ACTION _800_Reset:
Axis[ID].aStop();
CASE RestStep OF
0:(***************复位命令**************************)
	IF GVL_API.stAxis[ID].reset OR GVL.Reset THEN
		GVL_API.stAxis[ID].initialize:=FALSE;
		GVL_API.stAxis[ID].homeExe:=FALSE; 
		GVL_API.stAxis[ID].stop:=FALSE;
		GVL_API.stAxis[ID].JogBackwards:=FALSE;
		GVL_API.stAxis[ID].JogForward:=FALSE;
		GVL_API.stAxis[ID].MoveAbsoluteExe:=FALSE;
		GVL_API.stAxis[ID].MoveConstantVelocity:=FALSE;
		GVL_API.stAxis[ID].MoveRelativeExe:=FALSE;
		GVL_API.stAxis[ID].velocity:=0;
		GVL_API.stAxis[ID].requestedoffset:=0;
		GVL_API.stAxis[ID].requestedposition:=0;
		GVL_API.stAxis[ID].constantvelocitystart:=0;
		GVL_API.stAxis[ID].constanvelocityend:=0;
		FB_Home(ref:=Axis[ID].Ref , Execute:= FALSE);
		GVL_API.stAxis[ID].Home_Done:=FALSE;
		GVL_API.stAxis[ID].Move_Done:=FALSE;
		RestStep:=1;
	END_IF
1:	
		RestStep:=2;

2:(***************EORROR来的错误**************************)
		GVL_API.stAxis[ID].reset:=FALSE;
		parameter_out_of_range:=FALSE;
		SpeedNotReach:=FALSE;		
		RestStep:=20;
	
10:	(***************轴错误复位**************************)		
		Axis[ID].Reset_do:=TRUE;		
		RestStep:=100;		
20:	(***************轴停止*****************************)
		Axis[ID].aStop(stop_do:=TRUE);		
		RestStep:=30;
30:
	IF  Axis[ID].Ref.Status.NotMoving   THEN 		
		RestStep:=10;	
	END_IF
100:		
	IF Axis[ID].Ref.Status.NotMoving THEN 
		Axis[Id].aPower(power_do:=FALSE);
		GVL_API.stAxis[ID].Error:=FALSE;
		GVL_API.stAxis[ID].state:=AxisStateEnum.off;
		GVL_API.stAxis[ID].Errorid:=Axis_XY_ErrorEnum.no_error;
			SysStep:=0;
			RestStep:=0;
	END_IF
	  
END_CASE
END_ACTION

ACTION ACT_LOG:
(*************************LOG*******************************************)
log_ID:=100;
//initialize
AlarmActionArray[log_ID+1].AlarmMsg.EN	:=	'Fast Scan Initialize cmdtimeout:';
AlarmActionArray[log_ID+1].AlarmMsg.EN	:=CONCAT(AlarmActionArray[log_ID+1].AlarmMsg.EN,
																	LREAL_TO_STRING(GVL_API.stAxis[ID].commandtimeout));
AlarmActionArray[log_ID+1].AlarmMsg.EN	:=CONCAT(AlarmActionArray[log_ID+1].AlarmMsg.EN,'; velocity:');
AlarmActionArray[log_ID+1].AlarmMsg.EN	:=CONCAT(AlarmActionArray[log_ID+1].AlarmMsg.EN,
																	LREAL_TO_STRING(GVL_API.stAxis[ID].velocity));	
AlarmActionArray[log_ID+1].AlarmMsg.EN	:=CONCAT(AlarmActionArray[log_ID+1].AlarmMsg.EN,'; acce:');																
AlarmActionArray[log_ID+1].AlarmMsg.EN	:=CONCAT(AlarmActionArray[log_ID+1].AlarmMsg.EN,
																	LREAL_TO_STRING(GVL_API.stAxis[ID].acceleration));
AlarmActionArray[log_ID+1].AlarmMsg.EN	:=CONCAT(AlarmActionArray[log_ID+1].AlarmMsg.EN,'; maxposition:');	
AlarmActionArray[log_ID+1].AlarmMsg.EN	:=CONCAT(AlarmActionArray[log_ID+1].AlarmMsg.EN,
																	LREAL_TO_STRING(GVL_API.stAxis[ID].maxDistance));
fbSetAlarm[log_ID+1](
	InUse:=TRUE , 
	//EventId:=log_ID+1 , 
	EventActive:=GVL_API.stAxis[ID].initialize , 
	EventClass:=Alm_EventClass.Event , 
	ToTheLogFile:=TRUE, 
	ToTheHistory:=TRUE , 
 );
 //home
AlarmActionArray[log_ID+2].AlarmMsg.EN	:=	'Fast Scan Home homingvelocity:';
AlarmActionArray[log_ID+2].AlarmMsg.EN	:=CONCAT(AlarmActionArray[log_ID+2].AlarmMsg.EN,
																	LREAL_TO_STRING(GVL_API.stAxis[ID].homingvelocity));
AlarmActionArray[log_ID+2].AlarmMsg.EN	:=CONCAT(AlarmActionArray[log_ID+2].AlarmMsg.EN,'; homeoffset:');
AlarmActionArray[log_ID+2].AlarmMsg.EN	:=CONCAT(AlarmActionArray[log_ID+2].AlarmMsg.EN,
																	LREAL_TO_STRING(GVL_API.stAxis[ID].homeoffset));		
AlarmActionArray[log_ID+2].AlarmMsg.EN	:=CONCAT(AlarmActionArray[log_ID+2].AlarmMsg.EN,'; homingtimeout:');
AlarmActionArray[log_ID+2].AlarmMsg.EN	:=CONCAT(AlarmActionArray[log_ID+2].AlarmMsg.EN,
																	LREAL_TO_STRING(GVL_API.stAxis[ID].homingtimeout));																
fbSetAlarm[log_ID+2](
	InUse:=TRUE , 
	//EventId:=log_ID+2 , 
	EventActive:=GVL_API.stAxis[ID].homeExe , 
	EventClass:=Alm_EventClass.Event , 
	ToTheLogFile:=TRUE, 
	ToTheHistory:=TRUE , 
 );
 //MoveRelative
AlarmActionArray[log_ID+3].AlarmMsg.EN	:=CONCAT('Fast Scan MoveRelative displacement:',
																	LREAL_TO_STRING(GVL_API.stAxis[ID].requestedoffset));
AlarmActionArray[log_ID+3].AlarmMsg.EN	:=CONCAT(AlarmActionArray[log_ID+3].AlarmMsg.EN,'; velocity:');
AlarmActionArray[log_ID+3].AlarmMsg.EN	:=CONCAT(AlarmActionArray[log_ID+3].AlarmMsg.EN,
																	LREAL_TO_STRING(GVL_API.stAxis[ID].velocity));
AlarmActionArray[log_ID+3].AlarmMsg.EN	:=CONCAT(AlarmActionArray[log_ID+3].AlarmMsg.EN,'; acc:');
AlarmActionArray[log_ID+3].AlarmMsg.EN	:=CONCAT(AlarmActionArray[log_ID+3].AlarmMsg.EN,
																	LREAL_TO_STRING(GVL_API.stAxis[ID].acceleration));
AlarmActionArray[log_ID+3].AlarmMsg.EN	:=CONCAT(AlarmActionArray[log_ID+3].AlarmMsg.EN,'; jerk:');																	
AlarmActionArray[log_ID+3].AlarmMsg.EN	:=CONCAT(AlarmActionArray[log_ID+3].AlarmMsg.EN,
																	LREAL_TO_STRING(GVL_API.stAxis[ID].jerk));
fbSetAlarm[log_ID+3](
	InUse:=TRUE , 
	//EventId:=log_ID+3 , 
	EventActive:=GVL_API.stAxis[ID].MoveRelativeExe , 
	EventClass:=Alm_EventClass.Event , 
	ToTheLogFile:=TRUE, 
	ToTheHistory:=TRUE , 
 );
 //MoveAbsoluteExe
AlarmActionArray[log_ID+4].AlarmMsg.EN	:=CONCAT('Fast Scan MoveAbsolute position:',
																	LREAL_TO_STRING(GVL_API.stAxis[ID].requestedposition));
AlarmActionArray[log_ID+4].AlarmMsg.EN	:=CONCAT(AlarmActionArray[log_ID+4].AlarmMsg.EN,'; velocity:');
AlarmActionArray[log_ID+4].AlarmMsg.EN	:=CONCAT(AlarmActionArray[log_ID+4].AlarmMsg.EN,
																	LREAL_TO_STRING(GVL_API.stAxis[ID].velocity));
AlarmActionArray[log_ID+4].AlarmMsg.EN	:=CONCAT(AlarmActionArray[log_ID+4].AlarmMsg.EN,'; acc:');
AlarmActionArray[log_ID+4].AlarmMsg.EN	:=CONCAT(AlarmActionArray[log_ID+4].AlarmMsg.EN,
																	LREAL_TO_STRING(GVL_API.stAxis[ID].acceleration));
AlarmActionArray[log_ID+4].AlarmMsg.EN	:=CONCAT(AlarmActionArray[log_ID+4].AlarmMsg.EN,'; jerk:');																	
AlarmActionArray[log_ID+4].AlarmMsg.EN	:=CONCAT(AlarmActionArray[log_ID+4].AlarmMsg.EN,
																	LREAL_TO_STRING(GVL_API.stAxis[ID].jerk));
fbSetAlarm[log_ID+4](
	InUse:=TRUE , 
	//EventId:=log_ID+4 , 
	EventActive:=GVL_API.stAxis[ID].MoveAbsoluteExe , 
	EventClass:=Alm_EventClass.Event , 
	ToTheLogFile:=TRUE, 
	ToTheHistory:=TRUE , 
 );
 //MoveConstantVelocity
AlarmActionArray[log_ID+5].AlarmMsg.EN	:=CONCAT('Fast Scan MoveConstantVelocity,',
																LREAL_TO_STRING(GVL_API.stAxis[ID].constantvelocitystart));
AlarmActionArray[log_ID+5].AlarmMsg.EN	:=CONCAT(AlarmActionArray[log_ID+5].AlarmMsg.EN,'->');
AlarmActionArray[log_ID+5].AlarmMsg.EN	:=CONCAT(AlarmActionArray[log_ID+5].AlarmMsg.EN,
																LREAL_TO_STRING(GVL_API.stAxis[ID].constanvelocityend));
AlarmActionArray[log_ID+5].AlarmMsg.EN	:=CONCAT(AlarmActionArray[log_ID+5].AlarmMsg.EN,'->');
AlarmActionArray[log_ID+5].AlarmMsg.EN	:=CONCAT(AlarmActionArray[log_ID+5].AlarmMsg.EN,
																LREAL_TO_STRING(GVL_API.stAxis[ID].requestedposition));
AlarmActionArray[log_ID+5].AlarmMsg.EN	:=CONCAT(AlarmActionArray[log_ID+5].AlarmMsg.EN,'; velocity:');
AlarmActionArray[log_ID+5].AlarmMsg.EN	:=CONCAT(AlarmActionArray[log_ID+5].AlarmMsg.EN,
																	LREAL_TO_STRING(GVL_API.stAxis[ID].velocity));
AlarmActionArray[log_ID+5].AlarmMsg.EN	:=CONCAT(AlarmActionArray[log_ID+5].AlarmMsg.EN,'; acc:');
AlarmActionArray[log_ID+5].AlarmMsg.EN	:=CONCAT(AlarmActionArray[log_ID+5].AlarmMsg.EN,
																	LREAL_TO_STRING(GVL_API.stAxis[ID].acceleration));
AlarmActionArray[log_ID+5].AlarmMsg.EN	:=CONCAT(AlarmActionArray[log_ID+5].AlarmMsg.EN,'; jerk:');																	
AlarmActionArray[log_ID+5].AlarmMsg.EN	:=CONCAT(AlarmActionArray[log_ID+5].AlarmMsg.EN,
																	LREAL_TO_STRING(GVL_API.stAxis[ID].jerk));
fbSetAlarm[log_ID+5](
	InUse:=TRUE , 
	//EventId:=log_ID+5 , 
	EventActive:=GVL_API.stAxis[ID].MoveConstantVelocity , 
	EventClass:=Alm_EventClass.Event , 
	ToTheLogFile:=TRUE, 
	ToTheHistory:=TRUE , 
 );
//stop
AlarmActionArray[log_ID+6].AlarmMsg.EN	:=	'Fast Scan MoveStop ';
fbSetAlarm[log_ID+6](
	InUse:=TRUE , 
	//EventId:=log_ID+6 , 
	EventActive:=GVL_API.stAxis[ID].stop , 
	EventClass:=Alm_EventClass.Event , 
	ToTheLogFile:=TRUE, 
	ToTheHistory:=TRUE , 
 );
 //enabled
AlarmActionArray[log_ID+7].AlarmMsg.EN	:=	'Fast Scan Enabled ';
fbSetAlarm[log_ID+7](
	InUse:=TRUE , 
	//EventId:=log_ID+7 , 
	EventActive:=GVL_API.stAxis[ID].enabled , 
	EventClass:=Alm_EventClass.Event , 
	ToTheLogFile:=TRUE, 
	ToTheHistory:=TRUE , 
 );
  //disable
AlarmActionArray[log_ID+8].AlarmMsg.EN	:=	'Fast Scan Disable ';
fbSetAlarm[log_ID+8](
	InUse:=TRUE , 
	//EventId:=log_ID+8 , 
	EventActive:=GVL_API.stAxis[ID].Disable , 
	EventClass:=Alm_EventClass.Event , 
	ToTheLogFile:=TRUE, 
	ToTheHistory:=TRUE , 
 );
//ERROR,log_ErrorEnum只能等于一个常数
CASE GVL_API.stAxis[ID].errorid  OF
0	:	log_ErrorEnum	:=	0	;
1	:	log_ErrorEnum	:=	1	;
2	:	log_ErrorEnum	:=	2	;
3	:	log_ErrorEnum	:=	3	;
4	:	log_ErrorEnum	:=	4	;
5	:	log_ErrorEnum	:=	5	;
6	:	log_ErrorEnum	:=	6	;
7	:	log_ErrorEnum	:=	7	;
8	:	log_ErrorEnum	:=	8	;
9	:	log_ErrorEnum	:=	9	;
10	:	log_ErrorEnum	:=	10	;
11	:	log_ErrorEnum	:=	11	;
12	:	log_ErrorEnum	:=	12	;
13	:	log_ErrorEnum	:=	13	;
14	:	log_ErrorEnum	:=	14	;
15	:	log_ErrorEnum	:=	15	;
16	:	log_ErrorEnum	:=	16	;
666	:	log_ErrorEnum	:=	666	;

END_CASE

AlarmActionArray[log_ID+9].AlarmMsg.EN	:=CONCAT('Fast Scan Error: ',TO_STRING(log_ErrorEnum));
fbSetAlarm[log_ID+9](
	InUse:=TRUE , 
//	EventId:=log_ID+9 , 
	EventActive:=GVL_API.stAxis[ID].errorid<>0 AND GVL_API.stAxis[ID].errorid<>666 , 
	EventClass:=Alm_EventClass.Alarm , 
	ToTheLogFile:=TRUE, 
	ToTheHistory:=TRUE , 
 );
 
//reset
AlarmActionArray[log_ID+10].AlarmMsg.EN	:=	'Fast Scan Reset ';
fbSetAlarm[log_ID+10](
	InUse:=TRUE , 
	EventId:=log_ID+10 , 
	EventActive:=GVL_API.stAxis[ID].reset , 
	EventClass:=Alm_EventClass.Event , 
	ToTheLogFile:=TRUE, 
	ToTheHistory:=TRUE , 
 );
 //AXIX_ERRORID
 AlarmActionArray[log_ID+11].AlarmMsg.EN	:=CONCAT('Fast Scan Axis_ErrorID: ',
																		UDINT_TO_STRING(Axis[ID].Ref.Status.ErrorID));
fbSetAlarm[log_ID+11](
	InUse:=TRUE , 
	EventId:=log_ID+11 , 
	EventActive:=Axis[ID].Ref.Status.Error , 
	EventClass:=Alm_EventClass.Event , 
	ToTheLogFile:=TRUE, 
	ToTheHistory:=TRUE , 
 );
END_ACTION

ACTION ACT_Safety:
(*****************SAFETY******************************)
IF GVL_API.stAxis[ID].state<>AxisStateEnum.off AND  GVL_API.stAxis[ID].state<>AxisStateEnum.error THEN 
	IF GVl.Emstop_Button OR GVL.Emstop_SAFE  THEN 
		GVL_API.stAxis[ID].errorid:=Axis_XY_ErrorEnum.emergency_error;
		Axis[ID].aStop(stop_do:=TRUE,Dec:=HMI_EM_STOP_Dec_FS,Jerk:=HMI_EM_STOP_Jerk_FS);
		//Axis[ID].aStop(stop_do:=TRUE,Jerk:=GVL_API.stAxis[ID].jerk);
		SysStep:=700;
	ELSIF GVL.shuttle_crash OR  Axis[ID].IO.snLimitN OR Axis[ID].IO.snLimitP  THEN 	
		GVL_API.stAxis[ID].errorid:=Axis_XY_ErrorEnum.trigger_Limit;
		Axis[ID].aStop(stop_do:=TRUE,Dec:=HMI_EM_STOP_Dec_FS,Jerk:=HMI_EM_STOP_Jerk_FS);
		SysStep:=700;
	(*ELSIF GVL.interlock_triggered THEN 
		GVL_API.stAxis[ID].ErrorId:=Axis_XY_ErrorEnum.interlock_error;
		Axis[ID].aStop(stop_do:=TRUE,Dec:=HMI_EM_STOP_Dec_FS,Jerk:=HMI_EM_STOP_Jerk_FS);
		SysStep:=700;
	*)
	ELSIF  Axis[ID].mcReadStatus.ErrorID=18000 THEN 
		GVL_API.stAxis[ID].errorid:=Axis_XY_ErrorEnum.Drive_not_ready_for_operation;
		SysStep:=700;
	ELSIF   Axis[ID].mcReadStatus.ErrorID=17510 THEN 
		GVL_API.stAxis[ID].errorid:=Axis_XY_ErrorEnum.Invalid_IO_data_for_more_than_n_subsequent_NC_cycles_encoder;
		SysStep:=700;	
	ELSIF  Axis[ID].mcReadStatus.ErrorID<>0 THEN 
		GVL_API.stAxis[ID].errorid:=Axis[ID].mcReadStatus.ErrorID;
		SysStep:=700;
	//ELSE 
	//	GVL_API.stAxis[ID].error:=Axis_XY_ErrorEnum.no_error;
	//	SysStep:=700;			
	END_IF	
END_IF

(*****************AXIS_ERROR******************************)
GVL_API.stAxis[ID].AxisErrorId:=Axis[ID].Ref.Status.ErrorID;
END_ACTION

END_PROGRAM

// ---- POUs/010_Motion/MotionBase/FB_MoveFS_Exte.TcPOU
FUNCTION_BLOCK FB_MoveFS_Exte
VAR_INPUT
	enable	:BOOL;
	ref		:AXIS_REF;
	jogF	:BOOL;
	jogB	:BOOL;
	Move_Stop:BOOL;
	PosLimit			:BOOL;			(*正极限位信号*)
	NegLimit			:BOOL;			(*负极限位信号*)
	maxDistance			:LREAL;			(*最大行程*)
	Acceleration		:LREAL;
	Deceleration		:LREAL;
	Jerk				:LREAL;
END_VAR
VAR_OUTPUT	
END_VAR
VAR
	MC_Read:MC_ReadStatus;
	MC_ABS:MC_MoveAbsolute;
	MC_REL:MC_MoveRelative;
	MC_Jog:MC_Jog;
	
	MC_ABS1:MC_MoveAbsolute;

	step1,step2,step3		:INT;	
	R_TRIG1,R_TRIG2,R_TRIG3	:R_TRIG;
	R_TRIG_done				:R_TRIG;
	ton_NotMoving			:TON;
	ton_Moving				:TON;
	rel_do					:BOOL;
	abs_do					:BOOL;
	jogF_do					:BOOL;
	jogB_do					:BOOL;
	
	abs_do1    			    :BOOL;
	error					:BOOL;

	MoveAbsolute_Busy		:BOOL;
	MoveConstantVelocity_Busy:BOOL;
	MoveRelative_Busy		:BOOL;
	jog_EN					:BOOL;
	FB_START_r_trig:		R_TRIG;
	start					:BOOL;
	jog_f_trig				:F_TRIG;
	ton_NotMoving_r_trig:Tc2_Standard.R_TRIG;
	Positive_Direction:BOOL;//正向
	Negative_Direction:BOOL;//负向
	
END_VAR
VAR_IN_OUT 
	MoveRelExe					:BOOL;
	MoveAbsExe					:BOOL;
	MoveConstantVelocityExe		:BOOL;//
	Velo						:LREAL;	//mm/s
	TargetRel					:LREAL;//mm
	TargetAbs					:LREAL;//mm
	ConstantVelocityStart		:LREAL;//mm		The position to start moving with a constant velocity
												//      0 < ConstantVelocityStart< ConstanVelocityEnd< RequestedPosition
	ConstanVelocityEnd			:LREAL;//mm		The position to end moving with a constant velocity											
	Done						:BOOL;
	NotMovingTimeOut 			:BOOL;
	SpeedNotReach				:BOOL;
END_VAR

(*********************NOT MOVING TIMEOUT***************************)
FB_START_r_trig(CLK:=jogF OR jogB OR MoveRelExe OR MoveAbsExe OR MoveConstantVelocityExe  , Q=> );
IF FB_START_r_trig.Q THEN 
	start:=TRUE;
END_IF
ton_NotMoving(IN:=Ref.Status.NotMoving AND start  , PT:= T#5S, Q=> , ET=> );
ton_NotMoving_r_trig(CLK:=ton_NotMoving.Q , Q=> );
IF ton_NotMoving_r_trig.Q THEN 
		NotMovingTimeOut:=TRUE;	
END_IF

Call_FB();
JOG();
MoveAbsolute();
MoveConstantVelocity();
MoveRelative();


(*********************error***************************)
IF ton_NotMoving.Q OR error OR SpeedNotReach THEN	
	start:=FALSE;
	error:=FALSE;
	ton_NotMoving(IN:=FALSE);	
	step1:=step2:=step2:=0;	
	MoveRelExe:=FALSE;
	MoveAbsExe:=FALSE;
	MoveConstantVelocityExe:=FALSE;
	Velo:=0;
	TargetAbs:=0;
	TargetRel:=0;
	ConstantVelocityStart:=0;
	ConstanVelocityEnd:=0;
	step1:=step2:=step3:=0;
	R_TRIG1(CLK:=FALSE);
	R_TRIG2(CLK:=FALSE);
	R_TRIG3(CLK:=FALSE);
END_IF

(*********************move done***************************)
IF MoveAbsolute_Busy OR MoveConstantVelocity_Busy OR  MoveRelative_Busy THEN 
	Done:=FALSE;
	jogF:=FALSE;
	jogB:=FALSE;
END_IF

jog_f_trig(CLK:=jogB OR jogF , Q=> );

R_TRIG_done(CLK:=MC_REL.Done OR MC_ABS.Done OR MC_ABS1.Done  OR jog_f_trig.Q OR Move_Stop , Q=> );
IF R_TRIG_done.Q THEN 	
	start:=FALSE;
	R_TRIG_done(CLK:=FALSE);
	NotMovingTimeOut:=FALSE;
	ton_NotMoving(IN:=FALSE);
	step1:=step2:=step3:=0;	
	MoveRelExe:=FALSE;
	MoveAbsExe:=FALSE;
	MoveConstantVelocityExe:=FALSE;
	Velo:=0;
	TargetAbs:=0;
	TargetRel:=0;
	ConstantVelocityStart:=0;
	ConstanVelocityEnd:=0;
	Done:=TRUE ;
END_IF

ACTION Call_FB:
MC_Read(
	Axis:=ref , 
	Enable:=TRUE);
MC_REL(
	Axis:=ref , 
	Execute:=rel_do , 
	Distance:=TargetRel , 
	Velocity:=Velo , 
	Acceleration:=Acceleration , 
	Deceleration:=Deceleration , 
	Jerk:=Jerk , 
	BufferMode:= , 
	Options:= , 
	Done=> , 
	Busy=>MoveRelative_Busy , 
	Active=> , 
	CommandAborted=> , 
	Error=> , 
	ErrorID=> );
	IF MC_REL.Busy THEN 
		rel_do:=FALSE;
		MoveRelExe:=FALSE;
	END_IF
MC_ABS(
	Axis:=ref , 
	Execute:=abs_do , 
	Position:=TargetAbs , 
	Velocity:=Velo , 
	Acceleration:=Acceleration , 
	Deceleration:=Deceleration , 
	Jerk:=Jerk , 
	BufferMode:= , 
	Options:= , 
	Done=> , 
	Busy=>MoveAbsolute_Busy , 
	Active=> , 
	CommandAborted=> , 
	Error=> , 
	ErrorID=> );
	IF MC_ABS.Busy THEN 
		abs_do:=FALSE;
		MoveAbsExe:=FALSE;
	END_IF
MC_Jog(
	Axis:=ref , 
	JogForward:=jogF_do , 
	JogBackwards:=jogB_do , 
	Mode:=MC_JOGMODE_CONTINOUS , 
	Position:= , 
	Velocity:=Velo , 
	Acceleration:=Acceleration , 
	Deceleration:=Deceleration , 
	Jerk:=Jerk , 
	Done=> , 
	Busy=> , 
	Active=> , 
	CommandAborted=> , 
	Error=> , 
	ErrorID=> );
MC_ABS1(
	Axis:=ref , 
	Execute:=abs_do1 , 
	Position:=TargetAbs , 
	Velocity:=Velo , 
	Acceleration:=Acceleration , 
	Deceleration:=Deceleration , 
	Jerk:=Jerk , 
	BufferMode:= , 
	Options:= , 
	Done=> , 
	Busy=> , 
	Active=> , 
	CommandAborted=> , 
	Error=> , 
	ErrorID=> );
	IF MC_ABS1.Busy THEN 
		abs_do1:=FALSE;
		MoveConstantVelocityExe:=FALSE;
	END_IF
END_ACTION

ACTION JOG:
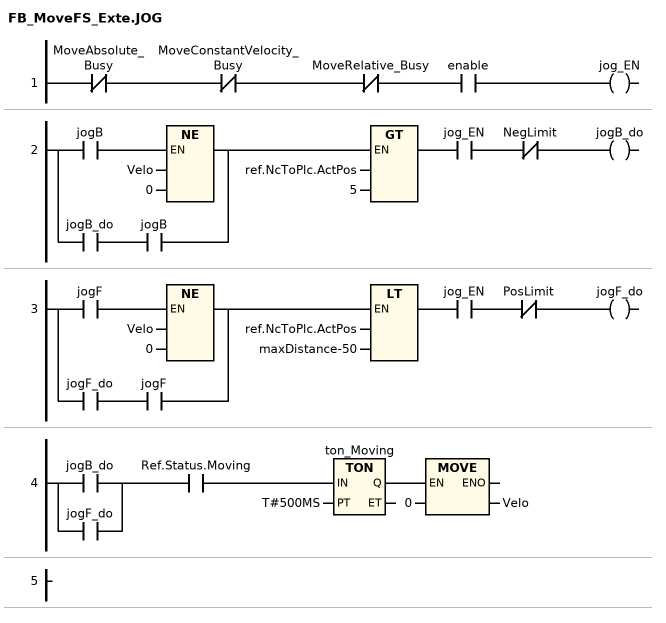
// NETWORK 1
jog_EN := NOT MoveAbsolute_Busy AND NOT MoveConstantVelocity_Busy AND NOT MoveRelative_Busy AND enable;

// NETWORK 2
jogB_do := ((jogB AND Velo <> 0 OR jogB_do AND jogB) AND ref.NcToPlc.ActPos > 5) AND jog_EN AND NOT NegLimit;

// NETWORK 3
jogF_do := ((jogF AND Velo <> 0 OR jogF_do AND jogF) AND ref.NcToPlc.ActPos < (maxDistance-50)) AND jog_EN AND NOT PosLimit;

// NETWORK 4
ton_Moving(IN := (jogB_do OR jogF_do) AND Ref.Status.Moving, PT := T#500MS); // TON
IF ton_Moving.Q THEN Velo := 0; END_IF

// NETWORK 5
END_ACTION

ACTION MoveAbsolute:
(****************ABS********************)
R_TRIG2(CLK:=MoveAbsExe AND Ref.Status.NotMoving AND enable   , Q=> );

CASE step2 OF 
	0:				
		IF R_TRIG2.Q THEN 
			R_TRIG2(CLK:=FALSE);			
			MoveAbsExe:=FALSE;
			step2:=1;
		END_IF
	1:	
		IF   Velo<>0 THEN 		
			abs_do:=TRUE;
			step2:=2;
		END_IF
	2:
		IF MC_ABS.Busy THEN 
			abs_do:=FALSE;								
			step2 :=0;
		END_IF	
END_CASE


IF  MoveAbsolute_Busy THEN 
	MoveRelExe:=FALSE;
	MoveConstantVelocityExe:=FALSE;
END_IF
END_ACTION

ACTION MoveConstantVelocity:
(****************MoveConstantVelocity********************)
R_TRIG3(CLK:=MoveConstantVelocityExe AND Ref.Status.NotMoving AND enable  , Q=> );
CASE step3 OF 
	0:				
		IF R_TRIG3.Q THEN 
			R_TRIG3(CLK:=FALSE);
			abs_do1:=FALSE;		
			MoveConstantVelocityExe:=FALSE;
			step3:=1;
		END_IF
	1:	//
		IF   Velo<>0 THEN 		
			abs_do1:=TRUE;
			step3:=2;
		END_IF
		
	2:	//启动第二段，匀速段,增加到达位置时速度判断
		IF ConstanVelocityEnd>ConstantVelocityStart THEN 
			Positive_Direction:=TRUE;
			Negative_Direction:=FALSE;
		ELSE
			Positive_Direction:=FALSE;
			Negative_Direction:=TRUE;	
		END_IF

			
		IF 	(Positive_Direction AND ref.NcToPlc.ActPos>=ConstantVelocityStart ) OR 
			(Negative_Direction AND ref.NcToPlc.ActPos<=ConstantVelocityStart ) THEN 
			
			 IF ABS(ABS(ref.NcToPlc.ActVelo)-Velo)<=30 THEN
				step3 :=3;
			 ELSE  
				step3 :=5;
			 END_IF
			
		END_IF
	3://满足第一段加速,检测减速度
		IF 	ABS(ref.NcToPlc.ActPos-ConstanVelocityEnd)<=30  THEN 
			IF ABS(ABS(ref.NcToPlc.ActVelo)-Velo)<=30 THEN
				step3 :=0;
			 ELSE  
				step3 :=5;
			 END_IF  
		END_IF	 
	5://ERROR
		SpeedNotReach:=TRUE;
		step3 :=0;
		
END_CASE
MoveConstantVelocity_Busy:=MC_ABS1.Busy ;

IF MoveConstantVelocity_Busy THEN 
	MoveRelExe:=FALSE;
	MoveAbsExe:=FALSE;
END_IF
END_ACTION

ACTION MoveRelative:
(****************Rel********************)
R_TRIG1(CLK:=MoveRelExe AND Ref.Status.NotMoving AND enable  , Q=> );
CASE step1 OF 
	0:				
		IF R_TRIG1.Q THEN 
			R_TRIG1(CLK:=FALSE);
			MoveRelExe:=FALSE;
			step1:=1;
		END_IF
	1:	
		IF TargetRel <>0 AND Velo<>0 THEN 		
			rel_do:=TRUE;
			step1:=2;
		END_IF
	2:
		IF MC_REL.Busy THEN 
			rel_do:=FALSE;								
			step1 :=0;
		END_IF	
END_CASE

IF MoveRelative_Busy THEN 
	MoveAbsExe:=FALSE;
	MoveConstantVelocityExe:=FALSE;
END_IF
END_ACTION

END_FUNCTION_BLOCK

// ---- POUs/010_Motion/MotionBase/FB_Home_X.TcPOU
FUNCTION_BLOCK FB_Home_X
(*========================================
Execute需一直有效，功能块才会一直执行
先回原点，然后直接到等待位
==========================================*)
VAR_IN_OUT
	ref				:AXIS_REF;	(* B *)
END_VAR
VAR_INPUT
	Execute				:BOOL;	(* B *)
	PosLimit			:BOOL;			(*正极限位信号*)
	NegLimit			:BOOL;			(*负极限位信号*)
	Position			:LREAL			(* B *) := DEFAULT_HOME_POSITION;
	HomeingVelo			:LREAL:=20;
	Standby_position	:LREAL;		//最终待机位
	bCalibrationCam 	:BOOL;	(* V *)	(* Beckhoff proprietary input *)
	rel_dis         	:LREAL:=50;  //碰到原点后，正向移动距离，在开始寻原点
	TimeOutSet       	:LREAL;//s
	reset				:BOOL;
END_VAR
VAR_OUTPUT
	Done				:BOOL;	(* B *)
	Busy				:BOOL;	(* E *)
	Active				:BOOL;	(* E *)
	CommandAborted		:BOOL;	(* E *)
	Error				:BOOL;	(* B *)
	ErrorID				:UDINT;	(* E *)
	TimeOut				:BOOL;
END_VAR
VAR
	mcJog			:MC_Jog;
	mcHome			:MC_Home;
	mcRel           :MC_MoveRelative;
	mcAbs           :MC_MoveAbsolute;	
	mcStop			:MC_Stop;
	HomeStep		:INT;
	ton				:TON;
	StopDo			:BOOL;
END_VAR

ton(IN:=Execute , PT:=LREAL_TO_TIME(TimeOutSet*1000) , Q=> , ET=> );
IF ton.Q THEN 
	TimeOut:=TRUE;
END_IF

IF  NOT Execute THEN
	mcJog.JogForward		:=FALSE;
	mcJog.JogBackwards		:=FALSE;
	mcHome.Execute			:=FALSE;
	mcRel.Execute			:=FALSE;
	mcAbs.Execute			:=FALSE;
	done					:=FALSE;
	busy					:=FALSE;	
	HomeStep				:=0;
END_IF

IF reset THEN 
	Error					:=FALSE;
	TimeOut					:=FALSE;
END_IF

CASE HomeStep OF

0:
	busy	:=FALSE;
	Done	:=FALSE;
	IF 	Execute AND NOT Error  THEN		
		IF  NOT bCalibrationCam THEN
			HomeStep	:=10;
		ELSE
			HomeStep	:=20;
		END_IF
		busy	:=TRUE;
		ErrorID	:=0;		
	END_IF
	
10:(*先向负限位方向运动*)
	mcJog.JogForward		:=FALSE;
	mcJog.JogBackwards		:=TRUE;		 
	IF	bCalibrationCam THEN
		mcJog.JogBackwards	:=FALSE;		 
		HomeStep	:=20;		
	ELSIF mcJog.Error OR TimeOut THEN
			HomeStep	:=100;
	END_IF
	
20:(*从原点处正方向移动一段距离*)
	mcRel.Execute		:=TRUE;	
	IF mcRel.Done AND ref.Status.NotMoving THEN 
		mcRel.Execute	:=FALSE;
		HomeStep		:=30;
	ELSIF mcRel.Error OR TimeOut THEN 
		HomeStep	:=100;	
	END_IF
	
30:(*调用回零功能块*)
	mcHome.Execute	:=TRUE;
	IF mcHome.Done AND ref.Status.Homed THEN
		mcHome.Execute	:=FALSE;		
		HomeStep		:=50;
	ELSIF ref.Status.Error OR TimeOut THEN
		HomeStep		:=100;
	END_IF
(*	
40:(*碰正极限*)
	mcJog.JogBackwards		:=FALSE;
	mcJog.JogForward		:=TRUE;		(*向正限位方向运动*)	
	IF PosLimit THEN 
		mcJog.JogForward	:=FALSE;
		IF Axis.Status.NotMoving THEN
			HomeStep	:=50;
		END_IF
	ELSIF mcJog.Error OR TimeOut THEN
			HomeStep	:=100; 
	END_IF
*)	
50:(*回待机位*)
	mcAbs.Execute:=TRUE;
	IF mcAbs.Done AND ref.Status.NotMoving THEN 
		mcAbs.Execute	:=FALSE;
		done			:=TRUE;
		HomeStep		:=99; 		
	END_IF
99:
	;	

100:
	Error			:=TRUE;
	IF	mcHome.ErrorID <> 0 THEN
		ErrorID			:=mcHome.ErrorID;
	ELSIF  mcJog.ErrorID <> 0 THEN
		ErrorID			:=mcJog.ErrorID;
	ELSIF mcRel.ErrorID<>0 THEN 
		ErrorID			:=mcRel.ErrorID;
	ELSIF mcAbs.ErrorID<>0 THEN 
		ErrorID			:=mcAbs.ErrorID;	
	END_IF
	mcJog.JogForward		:=FALSE;
	mcJog.JogBackwards		:=FALSE;
	mcHome.Execute			:=FALSE;
	mcRel.Execute			:=FALSE;
	mcAbs.Execute			:=FALSE;
	StopDo			:=TRUE;
	HomeStep		:=0;
	
END_CASE


Call_FB();

ACTION Call_FB:
ref.ReadStatus();
mcJog
	(
	Velocity:=	HomeingVelo ,
	Mode:=		MC_JOGMODE_CONTINOUS ,
	Axis:=		ref ,
	);

mcHome
	(
	Execute:= ,
	Position:=			Position ,
	HomingMode:= 		,
	BufferMode:= 		,
	Options:=			 ,
	bCalibrationCam:=	bCalibrationCam ,
	Axis:=				ref ,
	);

mcRel(
	Axis:=ref , 
	Execute:= , 
	Distance:=rel_dis , 
	Velocity:= HomeingVelo, 
	Acceleration:= , 
	Deceleration:= , 
	Jerk:= , 
	BufferMode:= , 
	Options:= , 
	Done=> , 
	Busy=> , 
	Active=> , 
	CommandAborted=> , 
	Error=> , 
	ErrorID=> );
mcAbs(
	Axis:=ref , 
	Execute:= , 
	Position:=Standby_position , 
	Velocity:=HomeingVelo , 
	Acceleration:= , 
	Deceleration:= , 
	Jerk:= , 
	BufferMode:= , 
	Options:= , 
	Done=> , 
	Busy=> , 
	Active=> , 
	CommandAborted=> , 
	Error=> , 
	ErrorID=> );
mcStop(
	Axis:=ref , 
	Execute:=StopDo , 
	Deceleration:= , 
	Jerk:= , 
	Options:= , 
	Done=> , 
	Busy=> , 
	Active=> , 
	CommandAborted=> , 
	Error=> , 
	ErrorID=> );
IF mcStop.Busy THEN 
	StopDo:=FALSE;
END_IF
END_ACTION

END_FUNCTION_BLOCK

// ---- POUs/010_Motion/YMove/P_SlowScan.TcPOU
PROGRAM P_SlowScan
VAR
	ID						:INT:=SlowScan;
	SysStep:				DINT;	
	HomeStep:				DINT;	
	RestStep				:DINT;
	MoveStep				:DINT;
	HomeDone:               BOOL;
	FB_move:				FB_MoveSS_Exte;
	FB_home:				FB_Home_X;
	ton_commandtimeout		:TON;
	
	ton1:Tc2_Standard.TON;
	Move_Done				:BOOL;
	NOT_Moving_TimeOut		:BOOL;
	parameter_out_of_range	:BOOL;
	actuator_out_of_pos_range:BOOL;
	actuator_out_of_neg_range:BOOL;	
	homeTimeOut				:BOOL;
	SpeedNotReach			:BOOL;	
	jog_EN					:BOOL;
	ton_Moving				:TON;
	log_ErrorEnum:Axis_XY_ErrorEnum;
	log_ID:INT;
END_VAR

ACT_LOG();
GVL_API.stAxis[ID].ControlLoopClosed:=Axis[ID].Ref.Status .ControlLoopClosed;
(*****************POS******************************)
GVL_API.stAxis[ID].position:=Axis[ID].Ref.NcToPlc.ActPos;

(*****************SysStep******************************)
CASE SysStep OF
0:	(*off*)
	_00_Waiting();				
100:(*idle*)		
	_100_Idle();								
200:(*home*)		
	_200_Homing();
300:(*ready*)	
	_300_Ready();							
400:(*disable*)	
	_400_Disable();			
500:(*Moving*)
	_500_Moving();	
600:(*Stopping*)
	_600_Stopping();
700:(*Error*)
	_700_Error();	
800:(*Reset*)
	_800_Reset();		
END_CASE
(*****************Reset*************************)
IF GVL_API.stAxis[ID].reset OR GVL.Reset THEN 
	SysStep:=800;	
END_IF

ACT_SAFETY();

Axis[ID].aReadStatus();
Axis[ID].aReset();

ACTION _00_Waiting:
IF GVL_API.stAxis[ID].initialize THEN 
	GVL_API.stAxis[ID].initialize:=FALSE;
	Axis[ID].aStop(stop_do:=TRUE);
	SysStep:=100;
ELSIF GVL_API.stAxis[ID].homeExe THEN 
	GVL_API.stAxis[ID].homeExe:=FALSE;  
	GVL_API.stAxis[ID].Home_Done:=TRUE;
	GVL_API.stAxis[ID].state:=AxisStateEnum.ready;	
	GVL_API.stAxis[ID].Home_Done:=FALSE;
	//SysStep:=200;
ELSIF GVL_API.stAxis[ID].MoveAbsoluteExe OR GVL_API.stAxis[ID].MoveRelativeExe 
		OR GVL_API.stAxis[ID].MoveVelocityExe OR GVL_API.stAxis[ID].JogBackwards 
		OR GVL_API.stAxis[ID].JogForward OR GVL_API.stAxis[ID].MoveConstantVelocity
		OR GVL_API.stAxis[ID].enabled OR GVL_API.stAxis[ID].Disable THEN 
	GVL_API.stAxis[ID].Move_Done:=FALSE;
	SysStep:=300;	
ELSIF GVL_API.stAxis[ID].stop THEN 
	SysStep:=600;	
ELSIF GVL_API.stAxis[ID].reset OR GVL.Reset THEN 
	SysStep:=800;	
END_IF


ton1(IN:=GVL_API.stAxis[ID].Home_Done OR  GVL_API.stAxis[ID].Move_Done , PT:=State_reset_time , Q=> , ET=> );
IF ton1.Q THEN 
	GVL_API.stAxis[ID].Home_Done:=FALSE;
	GVL_API.stAxis[ID].Move_Done:=FALSE;
END_IF
END_ACTION

ACTION _100_Idle:
Axis[ID].aStop(stop_do:=FALSE);
Axis[ID].aPower(power_do:=TRUE);	

IF axis[Id].Ref.Status .ControlLoopClosed THEN 
	//GVL_API.stAxis[ID].state:=AxisStateEnum.idle;//用原点命令
	GVL_API.stAxis[ID].state:=AxisStateEnum.ready;	//	无回原点命令
	GVL_API.stAxis[ID].Home_Done:=TRUE;//	无回原点命令
	SysStep :=0;
ELSIF GVl.Emstop_Button OR GVL.Emstop_SAFE THEN 
	GVL_API.stAxis[ID].errorid:=Axis_XY_ErrorEnum.emergency_error;
	SysStep:=700;
END_IF

(*******************commandtimeout*********************************)
ton_commandtimeout(IN:=NOT axis[Id].Ref.Status .ControlLoopClosed , 
	PT:=LREAL_TO_TIME(GVL_API.stAxis[ID].commandtimeout*1000) ,
	Q=> , ET=> );
IF ton_commandtimeout.Q  THEN 
	ton_commandtimeout(IN:=FALSE );
	GVL_API.stAxis[ID].errorid:=Axis_XY_ErrorEnum.cmd_timeout;
	SysStep:=700;	
END_IF

(*****************RESET******************************)
IF GVL_API.stAxis[ID].reset   THEN
	 SysStep:=800;
END_IF
END_ACTION

ACTION _200_Homing:
FB_Home(
		ref:=				Axis[ID].Ref , 
		Execute:= , 
		PosLimit:=			Axis[ID].IO.snLimitP , 
		Position:=			0 , 
		HomeingVelo:=		GVL_API.stAxis[ID].homingvelocity , 
		Standby_position:=  GVL_API.stAxis[ID].homeoffset,
		bCalibrationCam:=	Axis[ID].IO.snHome , 
		rel_dis:=			500 , 
		TimeOutSet:=		GVL_API.stAxis[ID].homingtimeout , 
		reset:= , 
		Done=> , 
		Busy=> , 
		Active=> , 
		CommandAborted=> , 
		Error=> , 
		ErrorID=> , 
		TimeOut=> );
		
CASE HomeStep OF
0:
	IF GVL_API.stAxis[ID].homingvelocity<>0 THEN 
		HomeStep:=10;
	END_IF
10:
	FB_Home.Execute:=TRUE;					
	IF FB_Home.Done THEN
		GVL_API.stAxis[ID].Home_Done:=TRUE;
		FB_Home.Execute:=FALSE;		
		HomeStep:=20;
	END_IF
	IF FB_Home.Error THEN 		
		GVL_API.stAxis[ID].ErrorId:=Axis_XY_ErrorEnum.homing_timeout;
		HomeStep:=30;
	END_IF
	
20:	(**********HOME DONE****************)
	
	GVL_API.stAxis[ID].state:=AxisStateEnum.ready;	
	HomeStep:=0;	
	SysStep:=0;
		
30:(**********TIME OUT****************)
	FB_Home.Execute:=FALSE;
	FB_Home.reset:=TRUE;
	HomeStep:=40;
40:(**********RESET****************)
	FB_Home.reset:=FALSE;
	HomeStep:=0;
	SysStep:=700;
		
END_CASE

IF FB_Home.Busy THEN 
	GVL_API.stAxis[ID].state:=AxisStateEnum.homing;
END_IF


(*****************RESET******************************)
IF GVL_API.stAxis[ID].reset   THEN
	FB_Home.Execute:=FALSE;
	 SysStep:=800;
END_IF
END_ACTION

ACTION _300_Ready:
Axis[ID].aStop();
GVL_API.stAxis[ID].Move_Done:=FALSE;
(*****************state******************************)
IF Axis[ID].Ref.Status.NotMoving AND axis[Id].Ref.Status .ControlLoopClosed  
AND NOT Axis[ID].Ref.Status.Error THEN 
	IF parameter_out_of_range THEN 
		GVL_API.stAxis[ID].errorid:=Axis_XY_ErrorEnum.parameter_out_of_range;
		SysStep:=700;
	ELSIF actuator_out_of_pos_range THEN 
		GVL_API.stAxis[ID].errorid:=Axis_XY_ErrorEnum.actuator_out_of_pos_range;
		SysStep:=700;
	ELSIF actuator_out_of_neg_range THEN 
		GVL_API.stAxis[ID].errorid:=Axis_XY_ErrorEnum.actuator_out_of_neg_range;
		SysStep:=700;	
	ELSE
		GVL_API.stAxis[ID].state:=AxisStateEnum.ready;
		GVL_API.stAxis[ID].errorid:=Axis_XY_ErrorEnum.no_error;
	END_IF
END_IF

(*****************valid command******************************)
IF NOT parameter_out_of_range 
AND axis[Id].Ref.Status .ControlLoopClosed  THEN  			
	IF GVL_API.stAxis[ID].MoveAbsoluteExe OR GVL_API.stAxis[ID].MoveRelativeExe 
		OR GVL_API.stAxis[ID].MoveVelocityExe OR GVL_API.stAxis[ID].JogBackwards 
		OR GVL_API.stAxis[ID].JogForward OR GVL_API.stAxis[ID].MoveConstantVelocity	THEN 	  		
			SysStep:=500;		
	END_IF
END_IF
(*****************enable-disable******************************)
IF GVL_API.stAxis[ID].enabled THEN 
	Axis[Id].aPower(power_do:=TRUE);	
	GVL_API.stAxis[ID].enabled:=FALSE;
	 GVL_API.stAxis[ID].state:=AxisStateEnum.ready;
	SysStep :=0;
ELSIF  GVL_API.stAxis[ID].Disable THEN 
	  SysStep:=400;
END_IF


(*****************RESET******************************)
IF GVL_API.stAxis[ID].reset THEN
	 SysStep:=800;
END_IF
END_ACTION

ACTION _400_Disable:
(*****************enable-disable******************************)
IF GVL_API.stAxis[ID].Disable THEN 
	Axis[Id].aPower(power_do:=FALSE);
	GVL_API.stAxis[ID].Disable:=FALSE;
	GVL_API.stAxis[ID].state:=AxisStateEnum.disabled;
	SysStep:=0;
END_IF

(*****************RESET******************************)
IF GVL_API.stAxis[ID].reset THEN
	 SysStep:=800;
END_IF
END_ACTION

ACTION _500_Moving:
IF Axis[ID].Ref.Status.Moving THEN 
	GVL_API.stAxis[ID].state:=AxisStateEnum.moving;
END_IF


IF NOT_Moving_TimeOut OR GVL_API.stAxis[ID].Move_Done  THEN 			(************NOT_Moving_TimeOut/Move_Done**************)
	NOT_Moving_TimeOut:=FALSE;	
	GVL_API.stAxis[ID].state:=AxisStateEnum.ready;			
	SysStep:=0;
ELSIF SpeedNotReach THEN 							(************SpeedNotReach**************)
	GVL_API.stAxis[ID].errorid:=Axis_XY_ErrorEnum.SpeedNotReach;
	SysStep:=700;
ELSIF Axis[ID].Ref.Status.NotMoving AND parameter_out_of_range THEN 
	GVL_API.stAxis[ID].errorid:=Axis_XY_ErrorEnum.parameter_out_of_range;
	SysStep:=700;
ELSIF Axis[ID].Ref.Status.Moving THEN 				(************trigger_limit**************)
	IF (Axis[ID].Ref.Status.NegativeDirection AND Axis[ID].IO.snHome) OR 
		(Axis[ID].Ref.Status.PositiveDirection AND Axis[ID].IO.snLimitP) 
		OR stInput.biElectromagnet_limit  OR stOutput.bqElectromagnet_power 
	THEN	
		Axis[ID].aStop(stop_do:=TRUE);
		GVL_API.stAxis[ID].errorid:=Axis_XY_ErrorEnum.trigger_limit;
		SysStep:=700;	
	END_IF 
	
ELSIF actuator_out_of_pos_range THEN 					(*********out_of_pos_range****************)
	Axis[ID].aStop(stop_do:=TRUE);
	GVL_API.stAxis[ID].errorid:=Axis_XY_ErrorEnum.actuator_out_of_pos_range;
	SysStep:=700;
ELSIF actuator_out_of_neg_range THEN
	Axis[ID].aStop(stop_do:=TRUE); 
	GVL_API.stAxis[ID].errorid:=Axis_XY_ErrorEnum.actuator_out_of_neg_range;
	SysStep:=700;	
ELSE GVL_API.stAxis[ID].errorid:=Axis_XY_ErrorEnum.no_error;
END_IF


(*****************JOG/ABS/REL/******************************)
(*****************MoveConstantVelocity*****************************)
IF NOT parameter_out_of_range  THEN 
	FB_move(
	enable:= 					NOT stInput.biElectromagnet_limit AND NOT stOutput.bqElectromagnet_power,	
	ref:= 						Axis[ID].Ref, 
	jogF:= 						GVL_API.stAxis[ID].JogForward, 
	jogB:= 						GVL_API.stAxis[ID].JogBackwards, 
	Acceleration:= 				GVL_API.stAxis[ID].acceleration, 
	Deceleration:= 				GVL_API.stAxis[ID].acceleration, 
	Jerk:= 						GVL_API.stAxis[ID].jerk, 	 
	MoveRelExe:= 				GVL_API.stAxis[ID].MoveRelativeExe, 
	MoveAbsExe:= 				GVL_API.stAxis[ID].MoveAbsoluteExe, 
	MoveConstantVelocityExe:= 	GVL_API.stAxis[ID].MoveConstantVelocity, 
	Velo:= 						GVL_API.stAxis[ID].velocity, 
	TargetRel:= 				GVL_API.stAxis[ID].requestedoffset, 
	TargetAbs:= 				GVL_API.stAxis[ID].requestedposition, 
	constantvelocityStart:= 	GVL_API.stAxis[ID].constantvelocitystart, 
	constanvelocityend:= 		GVL_API.stAxis[ID].constanvelocityend, 
	Done:= 						GVL_API.stAxis[ID].Move_Done,
	NotMovingTimeOut:= 			NOT_Moving_TimeOut,
	SpeedNotReach:=				SpeedNotReach
	);	
END_IF

(*****************stop******************************)
IF GVL_API.stAxis[ID].stop THEN 
	SysStep:=600;
END_IF
(*****************RESET******************************)
IF GVL_API.stAxis[ID].reset THEN
	 SysStep:=800;
END_IF
END_ACTION

ACTION _600_Stopping:
(**************只单独用作STOP命令*************************)
GVL_API.stAxis[ID].state:=AxisStateEnum.stopping;

Axis[ID].aStop(stop_do:=GVL_API.stAxis[ID].stop,Jerk:=GVL_API.stAxis[ID].jerk);
IF Axis[ID].mcStop.Busy THEN 
	GVL_API.stAxis[ID].state:=AxisStateEnum.stopping;	
	GVL_API.stAxis[ID].JogBackwards:=FALSE;
	GVL_API.stAxis[ID].JogForward:=FALSE;
	GVL_API.stAxis[ID].MoveAbsoluteExe:=FALSE;
	GVL_API.stAxis[ID].MoveConstantVelocity:=FALSE;
	GVL_API.stAxis[ID].MoveRelativeExe:=FALSE;
	GVL_API.stAxis[ID].velocity:=0;
	GVL_API.stAxis[ID].requestedoffset:=0;
	GVL_API.stAxis[ID].requestedposition:=0;
END_IF

IF Axis[ID].mcStop.Done AND Axis[ID].Ref.Status.NotMoving   THEN 		
	GVL_API.stAxis[ID].stop:=FALSE;
	GVL_API.stAxis[ID].state:=AxisStateEnum.ready;	
	GVL_API.stAxis[ID].Move_Done:=TRUE;
	SysStep:=0;
END_IF

(*****************RESET******************************)
IF GVL_API.stAxis[ID].reset THEN
	 GVL_API.stAxis[ID].stop:=FALSE;
	 Axis[ID].aStop(stop_do:=FALSE);
	 SysStep:=800;
END_IF
END_ACTION

ACTION _700_Error:
(*****************ERROR******************************)
GVL_API.stAxis[ID].Error:=TRUE;
GVL_API.stAxis[ID].state:=AxisStateEnum.error;
		GVL_API.stAxis[ID].initialize:=FALSE;
		GVL_API.stAxis[ID].homeExe:=FALSE; 
		GVL_API.stAxis[ID].stop:=FALSE;
		GVL_API.stAxis[ID].JogBackwards:=FALSE;
		GVL_API.stAxis[ID].JogForward:=FALSE;
		GVL_API.stAxis[ID].MoveAbsoluteExe:=FALSE;
		GVL_API.stAxis[ID].MoveConstantVelocity:=FALSE;
		GVL_API.stAxis[ID].MoveRelativeExe:=FALSE;
		GVL_API.stAxis[ID].velocity:=0;
		GVL_API.stAxis[ID].requestedoffset:=0;
		GVL_API.stAxis[ID].requestedposition:=0;
		GVL_API.stAxis[ID].constantvelocitystart:=0;
		GVL_API.stAxis[ID].constanvelocityend:=0;
		FB_Home.Execute:=FALSE;
		GVL_API.stAxis[ID].Home_Done:=FALSE;
		GVL_API.stAxis[ID].Move_Done:=FALSE;
 SysStep:=0;
END_ACTION

ACTION _800_Reset:
Axis[ID].aStop();
CASE RestStep OF
0:(***************复位命令**************************)
	IF GVL_API.stAxis[ID].reset OR GVL.Reset THEN
		GVL_API.stAxis[ID].initialize:=FALSE;
		GVL_API.stAxis[ID].homeExe:=FALSE; 
		GVL_API.stAxis[ID].stop:=FALSE;
		GVL_API.stAxis[ID].JogBackwards:=FALSE;
		GVL_API.stAxis[ID].JogForward:=FALSE;
		GVL_API.stAxis[ID].MoveAbsoluteExe:=FALSE;
		GVL_API.stAxis[ID].MoveConstantVelocity:=FALSE;
		GVL_API.stAxis[ID].MoveRelativeExe:=FALSE;
		GVL_API.stAxis[ID].velocity:=0;
		GVL_API.stAxis[ID].requestedoffset:=0;
		GVL_API.stAxis[ID].requestedposition:=0;
		GVL_API.stAxis[ID].constantvelocitystart:=0;
		GVL_API.stAxis[ID].constanvelocityend:=0;
		FB_Home.Execute:=FALSE;
		GVL_API.stAxis[ID].Home_Done:=FALSE;
		GVL_API.stAxis[ID].Move_Done:=FALSE;
		RestStep:=1;
	END_IF
1:	
		RestStep:=2;

2:(***************EORROR来的错误**************************)
		GVL_API.stAxis[ID].reset:=FALSE;
		parameter_out_of_range:=FALSE;
		SpeedNotReach:=FALSE;		
		RestStep:=20;
	
10:	(***************轴错误复位**************************)		
		Axis[ID].Reset_do:=TRUE;		
		RestStep:=100;		
20:	(***************轴停止*****************************)
		Axis[ID].aStop(stop_do:=TRUE);		
		RestStep:=30;
30:
	IF  Axis[ID].Ref.Status.NotMoving   THEN 		
		RestStep:=10;	
	END_IF
100:		
	IF Axis[ID].Ref.Status.NotMoving THEN 
		Axis[Id].aPower(power_do:=FALSE);
		GVL_API.stAxis[ID].Error:=FALSE;
		GVL_API.stAxis[ID].state:=AxisStateEnum.off;
		GVL_API.stAxis[ID].Errorid:=Axis_XY_ErrorEnum.no_error;
			SysStep:=0;
			RestStep:=0;
	END_IF
	  
END_CASE
END_ACTION

ACTION ACT_LOG:
(*************************LOG*******************************************)
log_ID:=130;
//initialize
AlarmActionArray[log_ID+1].AlarmMsg.EN	:=	'Slow Scan Initialize cmdtimeout: ';
AlarmActionArray[log_ID+1].AlarmMsg.EN	:=CONCAT(AlarmActionArray[log_ID+1].AlarmMsg.EN,
																	LREAL_TO_STRING(GVL_API.stAxis[ID].commandtimeout));
AlarmActionArray[log_ID+1].AlarmMsg.EN	:=CONCAT(AlarmActionArray[log_ID+1].AlarmMsg.EN,'; velocity:');
AlarmActionArray[log_ID+1].AlarmMsg.EN	:=CONCAT(AlarmActionArray[log_ID+1].AlarmMsg.EN,
																	LREAL_TO_STRING(GVL_API.stAxis[ID].velocity));	
AlarmActionArray[log_ID+1].AlarmMsg.EN	:=CONCAT(AlarmActionArray[log_ID+1].AlarmMsg.EN,'; acce:');																
AlarmActionArray[log_ID+1].AlarmMsg.EN	:=CONCAT(AlarmActionArray[log_ID+1].AlarmMsg.EN,
																	LREAL_TO_STRING(GVL_API.stAxis[ID].acceleration));
AlarmActionArray[log_ID+1].AlarmMsg.EN	:=CONCAT(AlarmActionArray[log_ID+1].AlarmMsg.EN,'; maxposition:');	
AlarmActionArray[log_ID+1].AlarmMsg.EN	:=CONCAT(AlarmActionArray[log_ID+1].AlarmMsg.EN,
																	LREAL_TO_STRING(GVL_API.stAxis[ID].maxDistance));
fbSetAlarm[log_ID+1](
	InUse:=TRUE , 
	EventId:=log_ID+1 , 
	EventActive:=GVL_API.stAxis[ID].initialize , 
	EventClass:=Alm_EventClass.Event , 
	ToTheLogFile:=TRUE, 
	ToTheHistory:=TRUE , 
 );

 //MoveRelative
AlarmActionArray[log_ID+3].AlarmMsg.EN	:=CONCAT('Slow Scan MoveRelative displacement:',
																	LREAL_TO_STRING(GVL_API.stAxis[ID].requestedoffset));
AlarmActionArray[log_ID+3].AlarmMsg.EN	:=CONCAT(AlarmActionArray[log_ID+3].AlarmMsg.EN,'; velocity:');
AlarmActionArray[log_ID+3].AlarmMsg.EN	:=CONCAT(AlarmActionArray[log_ID+3].AlarmMsg.EN,
																	LREAL_TO_STRING(GVL_API.stAxis[ID].velocity));
AlarmActionArray[log_ID+3].AlarmMsg.EN	:=CONCAT(AlarmActionArray[log_ID+3].AlarmMsg.EN,'; acc:');
AlarmActionArray[log_ID+3].AlarmMsg.EN	:=CONCAT(AlarmActionArray[log_ID+3].AlarmMsg.EN,
																	LREAL_TO_STRING(GVL_API.stAxis[ID].acceleration));
AlarmActionArray[log_ID+3].AlarmMsg.EN	:=CONCAT(AlarmActionArray[log_ID+3].AlarmMsg.EN,'; jerk:');																	
AlarmActionArray[log_ID+3].AlarmMsg.EN	:=CONCAT(AlarmActionArray[log_ID+3].AlarmMsg.EN,
																	LREAL_TO_STRING(GVL_API.stAxis[ID].jerk));
fbSetAlarm[log_ID+3](
	InUse:=TRUE , 
	EventId:=log_ID+3 , 
	EventActive:=GVL_API.stAxis[ID].MoveRelativeExe , 
	EventClass:=Alm_EventClass.Event , 
	ToTheLogFile:=TRUE, 
	ToTheHistory:=TRUE , 
 );
 //MoveAbsoluteExe
AlarmActionArray[log_ID+4].AlarmMsg.EN	:=CONCAT('Slow Scan MoveAbsolute position:',
																	LREAL_TO_STRING(GVL_API.stAxis[ID].requestedposition));
AlarmActionArray[log_ID+4].AlarmMsg.EN	:=CONCAT(AlarmActionArray[log_ID+4].AlarmMsg.EN,'; velocity:');
AlarmActionArray[log_ID+4].AlarmMsg.EN	:=CONCAT(AlarmActionArray[log_ID+4].AlarmMsg.EN,
																	LREAL_TO_STRING(GVL_API.stAxis[ID].velocity));
AlarmActionArray[log_ID+4].AlarmMsg.EN	:=CONCAT(AlarmActionArray[log_ID+4].AlarmMsg.EN,'; acc:');
AlarmActionArray[log_ID+4].AlarmMsg.EN	:=CONCAT(AlarmActionArray[log_ID+4].AlarmMsg.EN,
																	LREAL_TO_STRING(GVL_API.stAxis[ID].acceleration));
AlarmActionArray[log_ID+4].AlarmMsg.EN	:=CONCAT(AlarmActionArray[log_ID+4].AlarmMsg.EN,'; jerk:');																	
AlarmActionArray[log_ID+4].AlarmMsg.EN	:=CONCAT(AlarmActionArray[log_ID+4].AlarmMsg.EN,
																	LREAL_TO_STRING(GVL_API.stAxis[ID].jerk));

fbSetAlarm[log_ID+4](
	InUse:=TRUE , 
	EventId:=log_ID+4 , 
	EventActive:=GVL_API.stAxis[ID].MoveAbsoluteExe , 
	EventClass:=Alm_EventClass.Event , 
	ToTheLogFile:=TRUE, 
	ToTheHistory:=TRUE , 
 );

//stop
AlarmActionArray[log_ID+6].AlarmMsg.EN	:=	'Slow Scan MoveStop ';
fbSetAlarm[log_ID+6](
	InUse:=TRUE , 
	EventId:=log_ID+6 , 
	EventActive:=GVL_API.stAxis[ID].stop , 
	EventClass:=Alm_EventClass.Event , 
	ToTheLogFile:=TRUE, 
	ToTheHistory:=TRUE , 
 );
 //enabled
AlarmActionArray[log_ID+7].AlarmMsg.EN	:=	'Slow Scan Enabled ';
fbSetAlarm[log_ID+7](
	InUse:=TRUE , 
	EventId:=log_ID+7 , 
	EventActive:=GVL_API.stAxis[ID].enabled , 
	EventClass:=Alm_EventClass.Event , 
	ToTheLogFile:=TRUE, 
	ToTheHistory:=TRUE , 
 );
  //disable
AlarmActionArray[log_ID+8].AlarmMsg.EN	:=	'Slow Scan Disable ';
fbSetAlarm[log_ID+8](
	InUse:=TRUE , 
	EventId:=log_ID+8 , 
	EventActive:=GVL_API.stAxis[ID].Disable , 
	EventClass:=Alm_EventClass.Event , 
	ToTheLogFile:=TRUE, 
	ToTheHistory:=TRUE , 
 );
//ERROR,log_ErrorEnum只能等于一个常数
CASE GVL_API.stAxis[ID].errorid  OF
0	:	log_ErrorEnum	:=	0	;
1	:	log_ErrorEnum	:=	1	;
2	:	log_ErrorEnum	:=	2	;
3	:	log_ErrorEnum	:=	3	;
4	:	log_ErrorEnum	:=	4	;
5	:	log_ErrorEnum	:=	5	;
6	:	log_ErrorEnum	:=	6	;
7	:	log_ErrorEnum	:=	7	;
8	:	log_ErrorEnum	:=	8	;
9	:	log_ErrorEnum	:=	9	;
10	:	log_ErrorEnum	:=	10	;
11	:	log_ErrorEnum	:=	11	;
12	:	log_ErrorEnum	:=	12	;
13	:	log_ErrorEnum	:=	13	;
14	:	log_ErrorEnum	:=	14	;
15	:	log_ErrorEnum	:=	15	;
16	:	log_ErrorEnum	:=	16	;
666	:	log_ErrorEnum	:=	666	;

END_CASE

AlarmActionArray[log_ID+9].AlarmMsg.EN	:=CONCAT('Slow Scan Error: ',TO_STRING(log_ErrorEnum));
fbSetAlarm[log_ID+9](
	InUse:=TRUE , 
	EventId:=log_ID+9 , 
	EventActive:=GVL_API.stAxis[ID].error<>0 AND GVL_API.stAxis[ID].errorid<>666  , 
	EventClass:=Alm_EventClass.Alarm , 
	ToTheLogFile:=TRUE, 
	ToTheHistory:=TRUE , 
 );
 
//reset
AlarmActionArray[log_ID+10].AlarmMsg.EN	:=	'Slow Scan Reset ';
fbSetAlarm[log_ID+10](
	InUse:=TRUE , 
	EventId:=log_ID+10 , 
	EventActive:=GVL_API.stAxis[ID].reset , 
	EventClass:=Alm_EventClass.Event , 
	ToTheLogFile:=TRUE, 
	ToTheHistory:=TRUE , 
 );
  //AXIX_ERRORID
 AlarmActionArray[log_ID+11].AlarmMsg.EN	:=CONCAT('Slow Scan Axis_ErrorID: ',
																		UDINT_TO_STRING(Axis[ID].Ref.Status.ErrorID));
fbSetAlarm[log_ID+11](
	InUse:=TRUE , 
	EventId:=log_ID+11 , 
	EventActive:=Axis[ID].Ref.Status.Error , 
	EventClass:=Alm_EventClass.Event , 
	ToTheLogFile:=TRUE, 
	ToTheHistory:=TRUE , 
 );
END_ACTION

ACTION ACT_Safety:
(*****************SAFETY******************************)
IF GVL_API.stAxis[ID].state<>AxisStateEnum.off AND GVL_API.stAxis[ID].state<>AxisStateEnum.error THEN 
	IF GVl.Emstop_Button OR GVL.Emstop_SAFE  THEN 
		GVL_API.stAxis[ID].errorid:=Axis_XY_ErrorEnum.emergency_error;
		Axis[ID].aStop(stop_do:=TRUE,Jerk:=GVL_API.stAxis[ID].jerk);
		SysStep:=700;
	ELSIF GVL.shuttle_crash   THEN 	
		GVL_API.stAxis[ID].errorid:=Axis_XY_ErrorEnum.trigger_Limit;
		Axis[ID].aStop(stop_do:=TRUE,Jerk:=GVL_API.stAxis[ID].jerk);
		SysStep:=700;
	(*ELSIF GVL.interlock_triggered THEN 
		GVL_API.stAxis[ID].ErrorId:=Axis_XY_ErrorEnum.trigger_Limit;
		Axis[ID].aStop(stop_do:=TRUE,Jerk:=GVL_API.stAxis[ID].jerk);
		SysStep:=700;
	*)
	ELSIF   Axis[ID].mcReadStatus.ErrorID=18000 THEN 
		GVL_API.stAxis[ID].errorid:=Axis_XY_ErrorEnum.Drive_not_ready_for_operation;
		SysStep:=700;
	ELSIF   Axis[ID].mcReadStatus.ErrorID=17510 THEN 
		GVL_API.stAxis[ID].errorid:=Axis_XY_ErrorEnum.Invalid_IO_data_for_more_than_n_subsequent_NC_cycles_encoder;
		SysStep:=700;			
	ELSIF  Axis[ID].mcReadStatus.ErrorID<>0 THEN 
		GVL_API.stAxis[ID].errorid:=Axis[ID].mcReadStatus.ErrorID;
		SysStep:=700;
	//ELSE 
	//	GVL_API.stAxis[ID].error:=Axis_XY_ErrorEnum.no_error;	 
	//	SysStep:=700;
	END_IF
END_IF

(*****************AXIS_ERROR******************************)
GVL_API.stAxis[ID].AxisErrorId:=Axis[ID].Ref.Status.ErrorID;
END_ACTION

END_PROGRAM

// ---- POUs/010_Motion/MotionBase/FB_MoveSS_Exte.TcPOU
FUNCTION_BLOCK FB_MoveSS_Exte
VAR_INPUT
	enable	:BOOL;
	ref		:AXIS_REF;
	jogF	:BOOL;
	jogB	:BOOL;
	Acceleration		:LREAL;
	Deceleration		:LREAL;
	Jerk				:LREAL;
END_VAR
VAR_OUTPUT	
END_VAR
VAR
	MC_Read:MC_ReadStatus;
	MC_ABS:MC_MoveAbsolute;
	MC_REL:MC_MoveRelative;
	MC_Jog:MC_Jog;
	
	MC_ABS1:MC_MoveAbsolute;
	MC_ABS2:MC_MoveAbsolute;
	MC_VELO:MC_MoveVelocity;
	
	step1,step2,step3		:INT;	
	R_TRIG1,R_TRIG2,R_TRIG3	:R_TRIG;
	R_TRIG_done				:R_TRIG;
	ton_NotMoving			:TON;
	ton_Moving				:TON;
	rel_do					:BOOL;
	abs_do					:BOOL;
	jogF_do					:BOOL;
	jogB_do					:BOOL;
	
	abs_do1,abs_do2,velo_do	:BOOL;
	error					:BOOL;

	MoveAbsolute_Busy		:BOOL;
	MoveConstantVelocity_Busy:BOOL;
	MoveRelative_Busy		:BOOL;
	jog_EN					:BOOL;
	FB_START_r_trig:		R_TRIG;
	start					:BOOL;
	jog_f_trig				:F_TRIG;
	ton_NotMoving_r_trig:Tc2_Standard.R_TRIG;
END_VAR
VAR_IN_OUT 
	MoveRelExe					:BOOL;
	MoveAbsExe					:BOOL;
	MoveConstantVelocityExe		:BOOL;//
	Velo						:LREAL;	//mm/s
	TargetRel					:LREAL;//mm
	TargetAbs					:LREAL;//mm
	constantvelocityStart		:LREAL;//mm		The position to start moving with a constant velocity
												//      0 < ConstantVelocityStart< ConstanVelocityEnd< RequestedPosition
	constanvelocityEnd			:LREAL;//mm		The position to end moving with a constant velocity											
	Done						:BOOL;
	NotMovingTimeOut 			:BOOL;
	SpeedNotReach				:BOOL;
END_VAR

(*********************NOT MOVING TIMEOUT***************************)
FB_START_r_trig(CLK:=jogF OR jogB OR MoveRelExe OR MoveAbsExe OR MoveConstantVelocityExe  , Q=> );
IF FB_START_r_trig.Q THEN 
	start:=TRUE;
END_IF
ton_NotMoving(IN:=Ref.Status.NotMoving AND start  , PT:= T#5S, Q=> , ET=> );
ton_NotMoving_r_trig(CLK:=ton_NotMoving.Q , Q=> );
IF ton_NotMoving_r_trig.Q THEN 
		NotMovingTimeOut:=TRUE;	
END_IF

Call_FB();
JOG();
MoveAbsolute();
MoveConstantVelocity();
MoveRelative();


(*********************error***************************)
IF ton_NotMoving.Q OR error OR SpeedNotReach THEN	
	start:=FALSE;
	error:=FALSE;
	ton_NotMoving(IN:=FALSE);	
	step1:=step2:=step2:=0;	
	MoveRelExe:=FALSE;
	MoveAbsExe:=FALSE;
	MoveConstantVelocityExe:=FALSE;
	Velo:=0;
	TargetAbs:=0;
	TargetRel:=0;
	constantvelocityStart:=0;
	constanvelocityend:=0;
	step1:=step2:=step3:=0;
	R_TRIG1(CLK:=FALSE);
	R_TRIG2(CLK:=FALSE);
	R_TRIG3(CLK:=FALSE);
END_IF

(*********************move done***************************)
IF MoveAbsolute_Busy OR MoveConstantVelocity_Busy OR  MoveRelative_Busy THEN 
	Done:=FALSE;
	jogF:=FALSE;
	jogB:=FALSE;
END_IF

jog_f_trig(CLK:=jogB OR jogF , Q=> );

R_TRIG_done(CLK:=MC_REL.Done OR MC_ABS.Done OR MC_ABS2.Done OR jog_f_trig.Q , Q=> );
IF R_TRIG_done.Q THEN 	
	start:=FALSE;
	R_TRIG_done(CLK:=FALSE);
	NotMovingTimeOut:=FALSE;
	ton_NotMoving(IN:=FALSE);
	step1:=step2:=step2:=0;	
	MoveRelExe:=FALSE;
	MoveAbsExe:=FALSE;
	MoveConstantVelocityExe:=FALSE;
	Velo:=0;
	TargetAbs:=0;
	TargetRel:=0;
	constantvelocityStart:=0;
	constanvelocityend:=0;
	Done:=TRUE ;
END_IF

ACTION Call_FB:
MC_Read(
	Axis:=ref , 
	Enable:=TRUE);
MC_REL(
	Axis:=ref , 
	Execute:=rel_do , 
	Distance:=TargetRel , 
	Velocity:=Velo , 
	Acceleration:=Acceleration , 
	Deceleration:=Deceleration , 
	Jerk:=Jerk , 
	BufferMode:= , 
	Options:= , 
	Done=> , 
	Busy=>MoveRelative_Busy , 
	Active=> , 
	CommandAborted=> , 
	Error=> , 
	ErrorID=> );
	IF MC_REL.Busy THEN 
		rel_do:=FALSE;
		MoveRelExe:=FALSE;
	END_IF
MC_ABS(
	Axis:=ref , 
	Execute:=abs_do , 
	Position:=TargetAbs , 
	Velocity:=Velo , 
	Acceleration:=Acceleration , 
	Deceleration:=Deceleration , 
	Jerk:=Jerk , 
	BufferMode:= , 
	Options:= , 
	Done=> , 
	Busy=>MoveAbsolute_Busy , 
	Active=> , 
	CommandAborted=> , 
	Error=> , 
	ErrorID=> );
	IF MC_ABS.Busy THEN 
		abs_do:=FALSE;
		MoveAbsExe:=FALSE;
	END_IF
MC_Jog(
	Axis:=ref , 
	JogForward:=jogF_do , 
	JogBackwards:=jogB_do , 
	Mode:=MC_JOGMODE_CONTINOUS , 
	Position:= , 
	Velocity:=Velo , 
	Acceleration:=Acceleration , 
	Deceleration:=Deceleration , 
	Jerk:=Jerk , 
	Done=> , 
	Busy=> , 
	Active=> , 
	CommandAborted=> , 
	Error=> , 
	ErrorID=> );
MC_ABS1(
	Axis:=ref , 
	Execute:=abs_do1 , 
	Position:=constanvelocityend , 
	Velocity:=Velo , 
	Acceleration:=Acceleration , 
	Deceleration:=Deceleration , 
	Jerk:=Jerk , 
	BufferMode:= , 
	Options:= , 
	Done=> , 
	Busy=> , 
	Active=> , 
	CommandAborted=> , 
	Error=> , 
	ErrorID=> );
	IF MC_ABS1.Busy THEN 
		abs_do1:=FALSE;
		MoveConstantVelocityExe:=FALSE;
	END_IF
MC_VELO(
	Axis:=ref , 
	Execute:=velo_do , 
	Velocity:=Velo , 
	Acceleration:=Acceleration , 
	Deceleration:=Deceleration , 
	Jerk:=Jerk , 
	Direction:= , 
	BufferMode:= MC_Aborting, 
	Options:= , 
	InVelocity=> , 
	Busy=> , 
	Active=> , 
	CommandAborted=> , 
	Error=> , 
	ErrorID=> );
	//IF MC_VELO.Busy THEN 
	//	velo_do:=FALSE;
	//END_IF
MC_ABS2(
	Axis:=ref , 
	Execute:=abs_do2 , 
	Position:=TargetAbs , 
	Velocity:=Velo , 
	Acceleration:=Acceleration , 
	Deceleration:=Deceleration , 
	Jerk:=Jerk , 
	BufferMode:=MC_Aborting , 
	Options:= , 
	Done=> , 
	Busy=> , 
	Active=> , 
	CommandAborted=> , 
	Error=> , 
	ErrorID=> );
	IF MC_ABS2.Busy THEN 
		abs_do2:=FALSE;
	END_IF
END_ACTION

ACTION JOG:
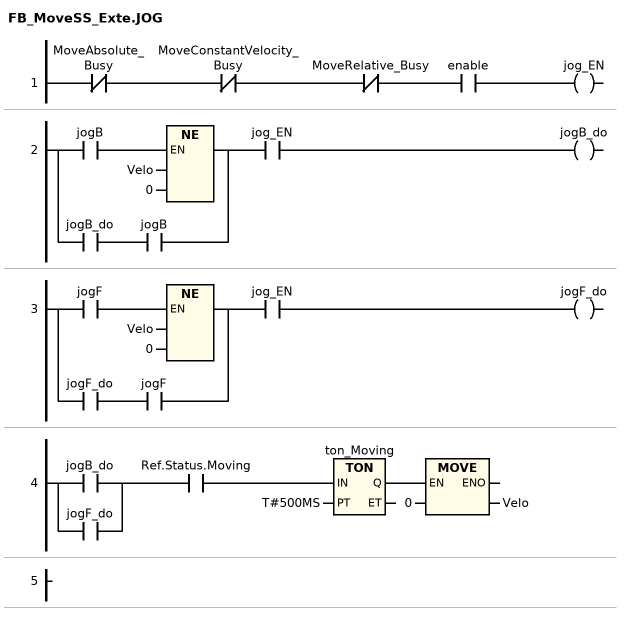
// NETWORK 1
jog_EN := NOT MoveAbsolute_Busy AND NOT MoveConstantVelocity_Busy AND NOT MoveRelative_Busy AND enable;

// NETWORK 2
jogB_do := (jogB AND Velo <> 0 OR jogB_do AND jogB) AND jog_EN;

// NETWORK 3
jogF_do := (jogF AND Velo <> 0 OR jogF_do AND jogF) AND jog_EN;

// NETWORK 4
ton_Moving(IN := (jogB_do OR jogF_do) AND Ref.Status.Moving, PT := T#500MS); // TON
IF ton_Moving.Q THEN Velo := 0; END_IF

// NETWORK 5
END_ACTION

ACTION MoveAbsolute:
(****************ABS********************)
R_TRIG2(CLK:=MoveAbsExe AND Ref.Status.NotMoving AND enable   , Q=> );

CASE step2 OF 
	0:				
		IF R_TRIG2.Q THEN 
			R_TRIG2(CLK:=FALSE);			
			MoveAbsExe:=FALSE;
			step2:=1;
		END_IF
	1:	
		IF   Velo<>0 THEN 		
			abs_do:=TRUE;
			step2:=2;
		END_IF
	2:
		IF MC_ABS.Busy THEN 
			abs_do:=FALSE;								
			step2 :=0;
		END_IF	
END_CASE


IF  MoveAbsolute_Busy THEN 
	MoveRelExe:=FALSE;
	MoveConstantVelocityExe:=FALSE;
END_IF
END_ACTION

ACTION MoveConstantVelocity:
(****************MoveConstantVelocity********************)
R_TRIG3(CLK:=MoveConstantVelocityExe AND Ref.Status.NotMoving AND enable  , Q=> );
CASE step3 OF 
	0:				
		IF R_TRIG3.Q THEN 
			R_TRIG3(CLK:=FALSE);
			MoveConstantVelocityExe:=FALSE;
			abs_do1:=abs_do2:=velo_do:=FALSE;		
			step3:=1;
		END_IF
	1:	//启动第一段，加速段
		IF   Velo<>0 THEN 		
			abs_do1:=TRUE;
			step3:=2;
		END_IF
		
	2:	//启动第二段，匀速段,增加到达位置时速度判断
		IF constanvelocityend>constantvelocityStart THEN 
			MC_VELO.Direction:=MC_Positive_Direction;
		ELSE
			MC_VELO.Direction:=MC_Negative_Direction;	
		END_IF
		
		IF 	(MC_VELO.Direction=MC_Positive_Direction AND ref.NcToPlc.ActPos>=constantvelocityStart)
			OR 	(MC_VELO.Direction=MC_Negative_Direction AND ref.NcToPlc.ActPos<=constantvelocityStart)  THEN 
			IF  ABS(ref.NcToPlc.ActVelo-velo)>10 THEN 
				abs_do1:=FALSE;	
				step3 :=5;
			END_IF
		END_IF
		
		IF ABS(ref.NcToPlc.ActVelo-velo)<=10 THEN			 
				abs_do1:=FALSE;					
				velo_do:=TRUE;									
				step3 :=3;
		END_IF
		
	3:	//启动第三段，减速段
		//IF MC_VELO.Busy THEN 
		//	velo_do:=FALSE;
		//END_IF
		IF (constanvelocityend>constantvelocityStart AND 
		 		ref.NcToPlc.ActPos>constanvelocityend)
		OR  (constanvelocityend<constantvelocityStart AND 
		 		ref.NcToPlc.ActPos<constanvelocityend)
		  THEN 	
			velo_do:=FALSE;
			abs_do2:=TRUE;
			step3 :=4;
		END_IF
	4:
		IF MC_ABS2.Busy THEN 
			abs_do2:=FALSE;
			step3 :=0;
		END_IF
	5://ERROR
		SpeedNotReach:=TRUE;
		step3 :=0;
		
END_CASE
MoveConstantVelocity_Busy:=MC_ABS1.Busy OR  MC_VELO.Busy OR MC_ABS2.Busy;

IF MoveConstantVelocity_Busy THEN 
	MoveRelExe:=FALSE;
	MoveAbsExe:=FALSE;
END_IF
END_ACTION

ACTION MoveConstantVelocity_old:
(****************MoveConstantVelocity********************)
R_TRIG3(CLK:=MoveConstantVelocityExe AND Ref.Status.NotMoving AND enable  , Q=> );
CASE step3 OF 
	0:				
		IF R_TRIG3.Q THEN 
			R_TRIG3(CLK:=FALSE);
			MoveConstantVelocityExe:=FALSE;
			abs_do1:=abs_do2:=velo_do:=FALSE;		
			step3:=1;
		END_IF
	1:	//启动第一段，加速段
		IF   Velo<>0 THEN 		
			abs_do1:=TRUE;
			step3:=2;
		END_IF
		
	2:	//启动第二段，匀速段,增加到达位置时速度判断
		IF constanvelocityend>constantvelocityStart THEN 
			MC_VELO.Direction:=MC_Positive_Direction;
		ELSE
			MC_VELO.Direction:=MC_Negative_Direction;	
		END_IF
		
		IF 	(MC_VELO.Direction=MC_Positive_Direction AND ref.NcToPlc.ActPos>=constantvelocityStart)
			OR 	(MC_VELO.Direction=MC_Negative_Direction AND ref.NcToPlc.ActPos<=constantvelocityStart)  THEN 
			IF NOT ref.Status.ConstantVelocity THEN 
				abs_do1:=FALSE;	
				step3 :=5;
			END_IF
		END_IF
		
		IF ref.Status.ConstantVelocity THEN			 
				abs_do1:=FALSE;					
				velo_do:=TRUE;									
				step3 :=3;
		END_IF
		
	3:	//启动第三段，减速段
		//IF MC_VELO.Busy THEN 
		//	velo_do:=FALSE;
		//END_IF
		IF (constanvelocityend>constantvelocityStart AND 
		 		ref.NcToPlc.ActPos>constanvelocityend)
		OR  (constanvelocityend<constantvelocityStart AND 
		 		ref.NcToPlc.ActPos<constanvelocityend)
		  THEN 	
			velo_do:=FALSE;
			abs_do2:=TRUE;
			step3 :=4;
		END_IF
	4:
		IF MC_ABS2.Busy THEN 
			abs_do2:=FALSE;
			step3 :=0;
		END_IF
	5://ERROR
		SpeedNotReach:=TRUE;
		step3 :=0;
		
END_CASE
MoveConstantVelocity_Busy:=MC_ABS1.Busy OR  MC_VELO.Busy OR MC_ABS2.Busy;

IF MoveConstantVelocity_Busy THEN 
	MoveRelExe:=FALSE;
	MoveAbsExe:=FALSE;
END_IF
END_ACTION

ACTION MoveRelative:
(****************Rel********************)
R_TRIG1(CLK:=MoveRelExe AND Ref.Status.NotMoving AND enable  , Q=> );
CASE step1 OF 
	0:				
		IF R_TRIG1.Q THEN 
			R_TRIG1(CLK:=FALSE);
			MoveRelExe:=FALSE;
			step1:=1;
		END_IF
	1:	
		IF TargetRel <>0 AND Velo<>0 THEN 		
			rel_do:=TRUE;
			step1:=2;
		END_IF
	2:
		IF MC_REL.Busy THEN 
			rel_do:=FALSE;								
			step1 :=0;
		END_IF	
END_CASE

IF MoveRelative_Busy THEN 
	MoveAbsExe:=FALSE;
	MoveConstantVelocityExe:=FALSE;
END_IF
END_ACTION

END_FUNCTION_BLOCK

// ---- POUs/010_Motion/ZMove/P_Z_Axis.TcPOU
PROGRAM P_Z_Axis
VAR
	ID						:INT:=Z_Axis;
	SysStep:				DINT;	
	HomeStep:				DINT;	
	RestStep				:DINT;
	MoveStep				:DINT;
	HomeDone:               BOOL;
	FB_move:				FB_MoveZ_Exte;
	FB_home:				FB_Home_Z;
	ton_commandtimeout		:TON;
	ton1:Tc2_Standard.TON;
	Move_Done				:BOOL;
	NOT_Moving_TimeOut		:BOOL;
	parameter_out_of_range	:BOOL;
	actuator_out_of_pos_range:BOOL;
	actuator_out_of_neg_range:BOOL;	
	homeTimeOut				:BOOL;
	SpeedNotReach			:BOOL;	
	jog_EN					:BOOL;
	ton_Moving				:TON;
	log_ErrorEnum:Axis_XY_ErrorEnum;
	log_ID:INT;

END_VAR

ACT_LOG();
GVL_API.stAxis[ID].ControlLoopClosed:=Axis[ID].Ref.Status .ControlLoopClosed;
GVL_API.stAxis[ID].jerk:=133;
(*****************POS******************************)
GVL_API.stAxis[ID].position:=Axis[ID].Ref.NcToPlc.ActPos;

(*****************SysStep******************************)
CASE SysStep OF
0:	(*off*)
	_00_Waiting();				
100:(*idle*)		
	_100_Idle();								
200:(*home*)		
	_200_Homing();
300:(*ready*)	
	_300_Ready();							
		
500:(*Moving*)
	_500_Moving();	
600:(*Stopping*)
	_600_Stopping();
700:(*Error*)
	_700_Error();	
800:(*Setoff*)
	_800_Setoff();	
END_CASE
(*****************Reset*************************)
IF GVL_API.stAxis[ID].reset OR GVL.Reset THEN 
	SysStep:=800;
    HomeStep:=0;	
END_IF

ACT_SAFETY();

Axis[ID].aReadStatus();
Axis[ID].aReset();

ACTION _00_Waiting:
IF GVL_API.stAxis[ID].initialize THEN 
	GVL_API.stAxis[ID].initialize:=FALSE;
	Axis[ID].aStop(stop_do:=TRUE);
	SysStep:=100;
ELSIF GVL_API.stAxis[ID].homeExe THEN 
	GVL_API.stAxis[ID].homeExe:=FALSE;  
	GVL_API.stAxis[ID].Home_Done:=FALSE;
	SysStep:=200;
ELSIF  GVL_API.stAxis[ID].MoveAbsoluteExe
		OR GVL_API.stAxis[ID].MoveRelativeExe
		OR GVL_API.stAxis[ID].Automatic_positioning  
		OR GVL_API.stAxis[ID].JogBackwards 
		OR GVL_API.stAxis[ID].JogForward THEN
	GVL_API.stAxis[ID].Move_Done:=FALSE;
	SysStep:=300;	
ELSIF GVL_API.stAxis[ID].stop THEN 
	SysStep:=600;	
ELSIF GVL_API.stAxis[ID].Setoff OR GVL.Reset THEN 
	SysStep:=800;	
END_IF

ton1(IN:=GVL_API.stAxis[ID].Home_Done OR  GVL_API.stAxis[ID].Move_Done , PT:=State_reset_time , Q=> , ET=> );
IF ton1.Q THEN 
	GVL_API.stAxis[ID].Home_Done:=FALSE;
	GVL_API.stAxis[ID].Move_Done:=FALSE;
END_IF
END_ACTION

ACTION _100_Idle:
Axis[ID].aStop(stop_do:=FALSE);
Axis[ID].aPower(power_do:=TRUE);	

IF axis[Id].Ref.Status .ControlLoopClosed THEN 
	GVL_API.stAxis[ID].state:=AxisStateEnum.idle;
	SysStep :=0;
ELSIF GVl.Emstop_Button OR GVL.Emstop_SAFE THEN 
	GVL_API.stAxis[ID].errorid:=Axis_XY_ErrorEnum.emergency_error;
	SysStep:=700;
END_IF

(*******************commandtimeout*********************************)
ton_commandtimeout(IN:=NOT axis[Id].Ref.Status .ControlLoopClosed , 
	PT:=LREAL_TO_TIME(GVL_API.stAxis[ID].commandtimeout*1000) ,
	Q=> , ET=> );
IF ton_commandtimeout.Q  THEN 
	ton_commandtimeout(IN:=FALSE );
	GVL_API.stAxis[ID].errorid:=Axis_XY_ErrorEnum.cmd_timeout;
	SysStep:=700;	
END_IF

(*****************RESET******************************)
IF GVL_API.stAxis[ID].reset   THEN
	 SysStep:=800;
END_IF
END_ACTION

ACTION _200_Homing:
stOutput.bqElectromagnet_power:=FALSE;
	FB_Home(
		Axis:=				Axis[ID].Ref , 
		Execute:= , 
		PosLimit:=			Axis[ID].IO.snLimitP OR Axis[ID].IO.snSpindle , 
		Position:=			0 , 
		HomeingVelo:=		GVL_API.stAxis[ID].homingvelocity , 
		Standby_position:=  0,
		bCalibrationCam:=	Axis[ID].IO.snHome , 
		rel_dis:=			10 , 
		TimeOutSet:=		GVL_API.stAxis[ID].homingtimeout , 
		reset:= ,
 		maxDistance:= GVL_API.stAxis[ID].maxDistance, 
		Done=> , 
		Busy=> , 
		Active=> , 
		CommandAborted=> , 
		Error=> , 
		ErrorID=> , 
		HomeErr=> , 
		TimeOut=>,
		 );

		
CASE HomeStep OF
0:
	IF GVL_API.stAxis[ID].homingvelocity<>0 THEN 
		HomeStep:=10;
	END_IF
10:
	FB_Home.Execute:=TRUE;					
	IF FB_Home.Done THEN
		GVL_API.stAxis[ID].Home_Done:=TRUE;
		FB_Home.Execute:=FALSE;	
		HomeStep:=20;
	END_IF
	
	IF FB_Home.TimeOut THEN 
		GVL_API.stAxis[ID].errorid:=Axis_Z_ErrorEnum.homing_timeout;
		HomeStep:=30;
	ELSIF FB_Home.HomeErr THEN 
		GVL_API.stAxis[ID].errorid:=Axis_Z_ErrorEnum.homing_error;
		HomeStep:=30;
	END_IF
	
20:	(**********HOME DONE****************)
	GVL_API.stAxis[ID].state:=AxisStateEnum.ready;	
	HomeStep:=0;	
	SysStep:=0;
30:(**********TIME OUT/error****************)
	FB_Home.Execute:=FALSE;
	FB_Home.reset:=TRUE;
	HomeStep:=40;
40:(**********RESET****************)
	FB_Home.reset:=FALSE;
	HomeStep:=0;
	SysStep:=700;
		
END_CASE

IF FB_Home.Busy THEN 
	GVL_API.stAxis[ID].state:=AxisStateEnum.homing;
END_IF
END_ACTION

ACTION _300_Ready:
Axis[ID].aStop();
GVL_API.stAxis[ID].Move_Done:=FALSE;
(***********parameter_out_of_range***********)
IF GVL_API.stAxis[ID].requestedposition>GVL_API.stAxis[ID].maxDistance OR GVL_API.stAxis[ID].requestedposition<0 THEN 
		parameter_out_of_range:=TRUE;
ELSE
		parameter_out_of_range:=FALSE;
END_IF	

(*********out_of_pos_range****************)
IF Axis[ID].Ref.NcToPlc.ActPos>GVL_API.stAxis[ID].maxDistance THEN 
	actuator_out_of_pos_range:=TRUE;
	actuator_out_of_neg_range:=FALSE;		
ELSIF	Axis[ID].Ref.NcToPlc.ActPos<-1 THEN 
	actuator_out_of_pos_range:=FALSE;
	actuator_out_of_neg_range:=TRUE;
ELSE
	actuator_out_of_pos_range:=FALSE;
	actuator_out_of_neg_range:=FALSE;
END_IF
	

(*****************state******************************)
IF Axis[ID].Ref.Status.NotMoving AND axis[Id].Ref.Status .ControlLoopClosed  
AND NOT Axis[ID].Ref.Status.Error THEN 
	IF parameter_out_of_range THEN 
		GVL_API.stAxis[ID].errorid:=Axis_Z_ErrorEnum.parameter_out_of_range;
		SysStep:=700;
	ELSIF actuator_out_of_pos_range THEN 
		GVL_API.stAxis[ID].errorid:=Axis_Z_ErrorEnum.actuator_out_of_pos_range;
		SysStep:=700;
	ELSIF actuator_out_of_neg_range THEN 
		GVL_API.stAxis[ID].errorid:=Axis_Z_ErrorEnum.actuator_out_of_neg_range;
		SysStep:=700;	
	ELSE
		GVL_API.stAxis[ID].state:=AxisStateEnum.ready;
		GVL_API.stAxis[ID].errorid:=Axis_Z_ErrorEnum.no_error;
	END_IF
END_IF

(*****************valid command******************************)
IF NOT parameter_out_of_range AND axis[Id].Ref.Status .ControlLoopClosed  THEN  			
	IF GVL_API.stAxis[ID].MoveAbsoluteExe
		OR GVL_API.stAxis[ID].MoveRelativeExe
		OR GVL_API.stAxis[ID].Automatic_positioning  
		OR GVL_API.stAxis[ID].JogBackwards 
		OR GVL_API.stAxis[ID].JogForward
		 
	THEN 	SysStep:=500;
	ELSIF GVL_API.stAxis[ID].homeExe  THEN			
			SysStep:=200;  	  							
	END_IF
END_IF

(*****************SETOFF******************************)
IF GVL_API.stAxis[ID].setoff THEN
	 SysStep:=800;
END_IF
END_ACTION

ACTION _500_Moving:
IF Axis[ID].Ref.Status.Moving THEN 
	GVL_API.stAxis[ID].state:=AxisStateEnum.moving;
END_IF

(*********out_of_pos_range****************)
IF Axis[ID].Ref.NcToPlc.ActPos>GVL_API.stAxis[ID].maxDistance THEN 
	actuator_out_of_pos_range:=TRUE;
	actuator_out_of_neg_range:=FALSE;
	GVL_API.stAxis[ID].JogForward:=FALSE;		
ELSIF	Axis[ID].Ref.NcToPlc.ActPos<-1 THEN 
	actuator_out_of_pos_range:=FALSE;
	actuator_out_of_neg_range:=TRUE;
	GVL_API.stAxis[ID].JogBackwards:=FALSE;
ELSE
	actuator_out_of_pos_range:=FALSE;
	actuator_out_of_neg_range:=FALSE;
END_IF

(*********parameter_out_of_range****************)
IF Axis[ID].IO.snHome 
	AND GVL_API.stAxis[ID].requestedposition<Axis[ID].Ref.NcToPlc.ActPos		
	THEN 	parameter_out_of_range:=TRUE;
ELSIF (Axis[ID].IO.snLimitP OR stInput.biElectromagnet_limit)
	AND  (GVL_API.stAxis[ID].requestedposition>Axis[ID].Ref.NcToPlc.ActPos
	OR 	GVL_API.stAxis[ID].requestedoffset>0)
	THEN 	parameter_out_of_range:=TRUE;
END_IF


IF NOT_Moving_TimeOut OR GVL_API.stAxis[ID].Move_Done  THEN 			(************NOT_Moving_TimeOut/Move_Done**************)
	NOT_Moving_TimeOut:=FALSE;	
	GVL_API.stAxis[ID].state:=AxisStateEnum.ready;			
	SysStep:=0;
ELSIF Axis[ID].Ref.Status.NotMoving AND parameter_out_of_range THEN 
	GVL_API.stAxis[ID].errorid:=Axis_Z_ErrorEnum.parameter_out_of_range;
	SysStep:=700;
ELSIF Axis[ID].Ref.Status.Moving THEN 				(************trigger_limit**************)
	IF (Axis[ID].Ref.Status.NegativeDirection AND Axis[ID].IO.snHome) OR 
		(Axis[ID].Ref.Status.PositiveDirection AND Axis[ID].IO.snLimitP)   
	THEN	
		Axis[ID].aStop(stop_do:=TRUE);
		GVL_API.stAxis[ID].errorid:=Axis_Z_ErrorEnum.trigger_limit;
		SysStep:=700;	
	END_IF 
	
ELSIF actuator_out_of_pos_range THEN 					(*********out_of_pos_range****************)
	Axis[ID].aStop(stop_do:=TRUE);
	GVL_API.stAxis[ID].errorid:=Axis_Z_ErrorEnum.actuator_out_of_pos_range;
	SysStep:=700;
ELSIF actuator_out_of_neg_range THEN
	Axis[ID].aStop(stop_do:=TRUE); 
	GVL_API.stAxis[ID].errorid:=Axis_Z_ErrorEnum.actuator_out_of_neg_range;
	SysStep:=700;	
ELSE GVL_API.stAxis[ID].errorid:=Axis_Z_ErrorEnum.no_error;
END_IF



IF NOT parameter_out_of_range THEN 
FB_move(
	ref:= Axis[ID].Ref, 
	jogF:= GVL_API.stAxis[ID].JogForward, 
	jogB:= GVL_API.stAxis[ID].JogBackwards, 
	PosLimit:= Axis[ID].IO.snLimitP, 
	NegLimit:= Axis[ID].IO.snHome, 
	electromagnetLimit:= stInput.biElectromagnet_limit, 
	maxDistance:= GVL_API.stAxis[ID].maxDistance, 
	Acceleration:= GVL_API.stAxis[ID].acceleration, 
	Deceleration:= GVL_API.stAxis[ID].acceleration, 
	Jerk:= GVL_API.stAxis[ID].jerk, 
	electromagnet_power=>stOutput.bqElectromagnet_power , 
	MoveRelExe:= GVL_API.stAxis[ID].MoveRelativeExe, 
	MoveAbsExe:= GVL_API.stAxis[ID].MoveAbsoluteExe, 
	MoveVelocityExe:=  GVL_API.stAxis[ID].Automatic_positioning, 
	Velo:= GVL_API.stAxis[ID].velocity, 
	TargetRel:=GVL_API.stAxis[ID].requestedoffset , 
	TargetAbs:= GVL_API.stAxis[ID].requestedposition, 
	Done:=GVL_API.stAxis[ID].Move_Done , 
	NotMovingTimeOut:= NOT_Moving_TimeOut);
END_IF

(*****************stop******************************)
IF GVL_API.stAxis[ID].stop THEN 
	SysStep:=600;
END_IF
END_ACTION

ACTION _600_Stopping:
(**************只单独用作STOP命令*************************)
GVL_API.stAxis[ID].state:=AxisStateEnum.stopping;

Axis[ID].aStop(stop_do:=GVL_API.stAxis[ID].stop,Jerk:=GVL_API.stAxis[ID].jerk);
IF Axis[ID].mcStop.Busy THEN 
	GVL_API.stAxis[ID].state:=AxisStateEnum.stopping;	
	GVL_API.stAxis[ID].JogBackwards:=FALSE;
	GVL_API.stAxis[ID].JogForward:=FALSE;
	GVL_API.stAxis[ID].MoveAbsoluteExe:=FALSE;
	GVL_API.stAxis[ID].requestedposition:=0;
END_IF

IF Axis[ID].mcStop.Done AND Axis[ID].Ref.Status.NotMoving   THEN 		
	GVL_API.stAxis[ID].stop:=FALSE;
	GVL_API.stAxis[ID].state:=AxisStateEnum.ready;	
	SysStep:=0;
END_IF
END_ACTION

ACTION _700_Error:
(*****************ERROR******************************)
GVL_API.stAxis[ID].Error:=TRUE;
GVL_API.stAxis[ID].state:=AxisStateEnum.error;
		GVL_API.stAxis[ID].initialize:=FALSE;
		GVL_API.stAxis[ID].homeExe:=FALSE; 
		GVL_API.stAxis[ID].stop:=FALSE;
		GVL_API.stAxis[ID].JogBackwards:=FALSE;
		GVL_API.stAxis[ID].JogForward:=FALSE;
		GVL_API.stAxis[ID].MoveAbsoluteExe:=FALSE;
		GVL_API.stAxis[ID].MoveRelativeExe:=FALSE;
		GVL_API.stAxis[ID].MoveVelocityExe:=FALSE;
		GVL_API.stAxis[ID].requestedposition:=0;
		GVL_API.stAxis[ID].requestedoffset:=0;			
		FB_Home.Execute:=FALSE;
 
SysStep:=0;
END_ACTION

ACTION _800_Setoff:
Axis[ID].aStop();
CASE RestStep OF
0:(***************复位命令**************************)
	IF GVL_API.stAxis[ID].setoff OR GVL.Reset THEN
		GVL_API.stAxis[ID].initialize:=FALSE;
		GVL_API.stAxis[ID].homeExe:=FALSE; 
		GVL_API.stAxis[ID].stop:=FALSE;
		GVL_API.stAxis[ID].JogBackwards:=FALSE;
		GVL_API.stAxis[ID].JogForward:=FALSE;
		GVL_API.stAxis[ID].MoveAbsoluteExe:=FALSE;
		GVL_API.stAxis[ID].MoveRelativeExe:=FALSE;
		GVL_API.stAxis[ID].MoveVelocityExe:=FALSE;
		GVL_API.stAxis[ID].requestedposition:=0;
		GVL_API.stAxis[ID].requestedoffset:=0;
		FB_Home( Axis:=Axis[ID].Ref ,Execute:=FALSE);
		RestStep:=1;
	END_IF
1:	
		RestStep:=2;

2:(***************EORROR来的错误**************************)
		GVL_API.stAxis[ID].Setoff:=FALSE;
		parameter_out_of_range:=FALSE;
		SpeedNotReach:=FALSE;		
		RestStep:=20;
	
10:	(***************轴错误复位**************************)		
		Axis[ID].Reset_do:=TRUE;		
		RestStep:=100;		
20:	(***************轴停止*****************************)
		Axis[ID].aStop(stop_do:=TRUE);		
		RestStep:=30;
30:
	IF  Axis[ID].Ref.Status.NotMoving   THEN 		
		RestStep:=10;	
	END_IF
100:		
	IF Axis[ID].Ref.Status.NotMoving THEN 
		Axis[Id].aPower(power_do:=FALSE);
		GVL_API.stAxis[ID].Error:=FALSE;
		GVL_API.stAxis[ID].state:=AxisStateEnum.off;
		GVL_API.stAxis[ID].Errorid:=Axis_XY_ErrorEnum.no_error;
			SysStep:=0;
			RestStep:=0;
	END_IF
	  
END_CASE
END_ACTION

ACTION ACT_LOG:
(*************************LOG*******************************************)
log_ID:=160;
//initialize
AlarmActionArray[log_ID+1].AlarmMsg.EN	:=	'Z_Axis initialize ';
AlarmActionArray[log_ID+1].AlarmMsg.EN	:=	'Z_Axis Initialize maxDistance:';
AlarmActionArray[log_ID+1].AlarmMsg.EN	:=CONCAT(AlarmActionArray[log_ID+1].AlarmMsg.EN,
																	LREAL_TO_STRING(GVL_API.stAxis[ID].maxDistance));
AlarmActionArray[log_ID+1].AlarmMsg.EN	:=CONCAT(AlarmActionArray[log_ID+1].AlarmMsg.EN,'; velocity:');
AlarmActionArray[log_ID+1].AlarmMsg.EN	:=CONCAT(AlarmActionArray[log_ID+1].AlarmMsg.EN,
																	LREAL_TO_STRING(GVL_API.stAxis[ID].velocity));	
AlarmActionArray[log_ID+1].AlarmMsg.EN	:=CONCAT(AlarmActionArray[log_ID+1].AlarmMsg.EN,'; acce:');																
AlarmActionArray[log_ID+1].AlarmMsg.EN	:=CONCAT(AlarmActionArray[log_ID+1].AlarmMsg.EN,
																	LREAL_TO_STRING(GVL_API.stAxis[ID].acceleration));

fbSetAlarm[log_ID+1](
	InUse:=TRUE , 
	EventId:=log_ID+1 , 
	EventActive:=GVL_API.stAxis[ID].initialize , 
	EventClass:=Alm_EventClass.Event , 
	ToTheLogFile:=TRUE, 
	ToTheHistory:=TRUE , 
 );
//home
AlarmActionArray[log_ID+2].AlarmMsg.EN	:=	'Z_Axis Home homingvelocity:';
AlarmActionArray[log_ID+2].AlarmMsg.EN	:=CONCAT(AlarmActionArray[log_ID+2].AlarmMsg.EN,
																	LREAL_TO_STRING(GVL_API.stAxis[ID].homingvelocity));
fbSetAlarm[log_ID+2](
	InUse:=TRUE , 
	EventId:=log_ID+2 , 
	EventActive:=GVL_API.stAxis[ID].homeExe , 
	EventClass:=Alm_EventClass.Event , 
	ToTheLogFile:=TRUE, 
	ToTheHistory:=TRUE , 
 );
 //MoveAbsoluteExe
AlarmActionArray[log_ID+4].AlarmMsg.EN	:=CONCAT('Z_Axis MoveAbsolute, position:',
																LREAL_TO_STRING(GVL_API.stAxis[ID].requestedposition));
AlarmActionArray[log_ID+4].AlarmMsg.EN	:=CONCAT(AlarmActionArray[log_ID+4].AlarmMsg.EN,', velocity:');
AlarmActionArray[log_ID+4].AlarmMsg.EN	:=CONCAT(AlarmActionArray[log_ID+4].AlarmMsg.EN,
																LREAL_TO_STRING(GVL_API.stAxis[ID].velocity));
fbSetAlarm[log_ID+4](
	InUse:=TRUE , 
	EventId:=log_ID+4 , 
	EventActive:=GVL_API.stAxis[ID].MoveAbsoluteExe , 
	EventClass:=Alm_EventClass.Event , 
	ToTheLogFile:=TRUE, 
	ToTheHistory:=TRUE , 
 );

//stop
AlarmActionArray[log_ID+6].AlarmMsg.EN	:=	'Z_Axis MoveStop ';
fbSetAlarm[log_ID+6](
	InUse:=TRUE , 
	EventId:=log_ID+6 , 
	EventActive:=GVL_API.stAxis[ID].stop , 
	EventClass:=Alm_EventClass.Event , 
	ToTheLogFile:=TRUE, 
	ToTheHistory:=TRUE , 
 );

//ERROR,log_ErrorEnum只能等于一个常数
CASE GVL_API.stAxis[ID].errorid  OF
0	:	log_ErrorEnum	:=	0	;
1	:	log_ErrorEnum	:=	1	;
2	:	log_ErrorEnum	:=	2	;
3	:	log_ErrorEnum	:=	3	;
4	:	log_ErrorEnum	:=	4	;
5	:	log_ErrorEnum	:=	5	;
6	:	log_ErrorEnum	:=	6	;
7	:	log_ErrorEnum	:=	7	;
8	:	log_ErrorEnum	:=	8	;
9	:	log_ErrorEnum	:=	9	;
10	:	log_ErrorEnum	:=	10	;
11	:	log_ErrorEnum	:=	11	;
12	:	log_ErrorEnum	:=	12	;
13	:	log_ErrorEnum	:=	13	;
14	:	log_ErrorEnum	:=	14	;
15	:	log_ErrorEnum	:=	15	;
666	:	log_ErrorEnum	:=	666	;

END_CASE

AlarmActionArray[log_ID+9].AlarmMsg.EN	:=CONCAT('Z_Axis Error: ',TO_STRING(log_ErrorEnum));
fbSetAlarm[log_ID+9](
	InUse:=TRUE , 
	EventId:=log_ID+9 , 
	EventActive:=GVL_API.stAxis[ID].error<>0 AND GVL_API.stAxis[ID].errorid<>666  , 
	EventClass:=Alm_EventClass.Alarm , 
	ToTheLogFile:=TRUE, 
	ToTheHistory:=TRUE , 
 );
 
//reset
AlarmActionArray[log_ID+10].AlarmMsg.EN	:=	'Z_Axis Reset ';
fbSetAlarm[log_ID+10](
	InUse:=TRUE , 
	EventId:=log_ID+10 , 
	EventActive:=GVL_API.stAxis[ID].setoff , 
	EventClass:=Alm_EventClass.Event , 
	ToTheLogFile:=TRUE, 
	ToTheHistory:=TRUE , 
 );
  //AXIX_ERRORID
 AlarmActionArray[log_ID+11].AlarmMsg.EN	:=CONCAT('Z_Axis Axis_ErrorID: ',
																		UDINT_TO_STRING(Axis[ID].Ref.Status.ErrorID));
fbSetAlarm[log_ID+11](
	InUse:=TRUE , 
	EventId:=log_ID+11 , 
	EventActive:=Axis[ID].Ref.Status.Error , 
	EventClass:=Alm_EventClass.Event , 
	ToTheLogFile:=TRUE, 
	ToTheHistory:=TRUE , 
 );
END_ACTION

ACTION ACT_Safety:
(*****************SAFETY******************************)
IF GVL_API.stAxis[ID].state<>AxisStateEnum.off AND GVL_API.stAxis[ID].state<>AxisStateEnum.error THEN 
	IF GVL.Emstop_Button   THEN 
		GVL_API.stAxis[ID].errorid:=Axis_Z_ErrorEnum.emergency_error;
		Axis[ID].aStop(stop_do:=TRUE,Jerk:=GVL_API.stAxis[ID].jerk);
		SysStep:=700;
	ELSIF   Axis[ID].mcReadStatus.ErrorID=18000 THEN 
		GVL_API.stAxis[ID].errorid:=Axis_XY_ErrorEnum.Drive_not_ready_for_operation;
		SysStep:=700;
	ELSIF   Axis[ID].mcReadStatus.ErrorID=17510 THEN 
		GVL_API.stAxis[ID].errorid:=Axis_XY_ErrorEnum.Invalid_IO_data_for_more_than_n_subsequent_NC_cycles_encoder;
		SysStep:=700;	
	ELSIF  Axis[ID].mcReadStatus.ErrorID<>0 THEN 
		GVL_API.stAxis[ID].errorid:=Axis[ID].mcReadStatus.ErrorID;
		SysStep:=700;
	//ELSE 
	//	GVL_API.stAxis[ID].error:=Axis_XY_ErrorEnum.no_error;	
	//	SysStep:=700;	
	END_IF
	
END_IF


IF GVL_API.stAxis[ID].state=AxisStateEnum.moving THEN 
	IF GVL.shuttle_crash OR  Axis[ID].IO.snLimitP THEN 	
		GVL_API.stAxis[ID].errorid:=Axis_Z_ErrorEnum.trigger_Limit;
		Axis[ID].aStop(stop_do:=TRUE,Jerk:=GVL_API.stAxis[ID].jerk);
		SysStep:=700;
	END_IF
END_IF
(*****************AXIS_ERROR******************************)
GVL_API.stAxis[ID].AxisErrorId:=Axis[ID].Ref.Status.ErrorID;
END_ACTION

END_PROGRAM

// ---- POUs/010_Motion/MotionBase/FB_MoveZ_Exte.TcPOU
FUNCTION_BLOCK FB_MoveZ_Exte
VAR_INPUT
	ref		:AXIS_REF;
	jogF	:BOOL;
	jogB	:BOOL;
	PosLimit			:BOOL;			(*正极限位信号*)
	NegLimit			:BOOL;			(*负极限位信号*)
	electromagnetLimit	:BOOL;
	
	maxDistance			:LREAL;			(*最大行程*)
	Acceleration		:LREAL;
	Deceleration		:LREAL;
	Jerk				:LREAL;
END_VAR
VAR_OUTPUT	
	electromagnet_power :BOOL;
END_VAR
VAR
	MC_Read:MC_ReadStatus;
	MC_ABS:MC_MoveAbsolute;
	MC_REL:MC_MoveRelative;
	MC_Jog:MC_Jog;	
	MC_VELO:MC_MoveVelocity;
	MC_stop:MC_Stop;
	
	step1,step2,step3		:INT;	
	R_TRIG1,R_TRIG2,R_TRIG3	:R_TRIG;
	R_TRIG_done				:R_TRIG;
	ton_NotMoving			:TON;
	ton_Moving				:TON;
	rel_do					:BOOL;
	abs_do					:BOOL;
	jogF_do					:BOOL;
	jogB_do					:BOOL;
	
	velo_do					:BOOL;
	stop_do					:BOOL;
	error					:BOOL;

	MoveAbsolute_Busy		:BOOL;
	MoveVelocity_Busy		:BOOL;
	MoveRelative_Busy		:BOOL;
	jog_EN					:BOOL;
	FB_START_r_trig:		R_TRIG;
	start					:BOOL;
	jog_f_trig				:F_TRIG;
END_VAR
VAR_IN_OUT 
	MoveRelExe					:BOOL;
	MoveAbsExe					:BOOL;
	MoveVelocityExe				:BOOL;//
	Velo						:LREAL;	//mm/s
	TargetRel					:LREAL;//mm
	TargetAbs					:LREAL;//mm
							
	Done						:BOOL;
	NotMovingTimeOut 			:BOOL;
	
END_VAR

(*********************NOT MOVING TIMEOUT***************************)
FB_START_r_trig(CLK:=jogF OR jogB OR MoveRelExe OR MoveAbsExe OR MoveVelocityExe  , Q=> );
IF FB_START_r_trig.Q THEN 
	start:=TRUE;
END_IF
ton_NotMoving(IN:=Ref.Status.NotMoving AND start  , PT:= T#5S, Q=> , ET=> );

Call_FB();
JOG();
MoveAbsolute();
MoveVelocity();
MoveRelative();


(*********************error***************************)
IF ton_NotMoving.Q OR error  THEN	
	start:=FALSE;
	NotMovingTimeOut:=TRUE;	
	error:=FALSE;
	ton_NotMoving(IN:=FALSE);	
	step1:=step2:=step2:=0;	
	MoveRelExe:=FALSE;
	MoveAbsExe:=FALSE;
	MoveVelocityExe:=FALSE;
	TargetAbs:=0;
	TargetRel:=0;
	

	R_TRIG1(CLK:=FALSE);
	R_TRIG2(CLK:=FALSE);
	R_TRIG3(CLK:=FALSE);
END_IF

(*********************move done***************************)
IF MoveAbsolute_Busy OR MoveVelocity_Busy OR  MoveRelative_Busy THEN 
	Done:=FALSE;
	jogF:=FALSE;
	jogB:=FALSE;
END_IF

jog_f_trig(CLK:=jogB OR jogF , Q=> );

R_TRIG_done(CLK:=MC_REL.Done OR MC_ABS.Done OR MC_stop.Done  OR jog_f_trig.Q , Q=> );
IF R_TRIG_done.Q THEN 	
	start:=FALSE;
	R_TRIG_done(CLK:=FALSE);
	NotMovingTimeOut:=FALSE;
	ton_NotMoving(IN:=FALSE);
	step1:=step2:=step2:=0;	
	MoveRelExe:=FALSE;
	MoveAbsExe:=FALSE;
	MoveVelocityExe:=FALSE;
	TargetAbs:=0;
	TargetRel:=0;
	
	Done:=TRUE ;
END_IF

ACTION Call_FB:
MC_Read(
	Axis:=ref , 
	Enable:=TRUE);
MC_REL(
	Axis:=ref , 
	Execute:=rel_do , 
	Distance:=TargetRel , 
	Velocity:=Velo , 
	Acceleration:=Acceleration , 
	Deceleration:=Deceleration , 
	Jerk:=Jerk , 
	BufferMode:= , 
	Options:= , 
	Done=> , 
	Busy=>MoveRelative_Busy , 
	Active=> , 
	CommandAborted=> , 
	Error=> , 
	ErrorID=> );
	IF MC_REL.Busy THEN 
		rel_do:=FALSE;
		MoveRelExe:=FALSE;
	END_IF
MC_ABS(
	Axis:=ref , 
	Execute:=abs_do , 
	Position:=TargetAbs , 
	Velocity:=Velo , 
	Acceleration:=Acceleration , 
	Deceleration:=Deceleration , 
	Jerk:=Jerk , 
	BufferMode:= , 
	Options:= , 
	Done=> , 
	Busy=>MoveAbsolute_Busy , 
	Active=> , 
	CommandAborted=> , 
	Error=> , 
	ErrorID=> );
	IF MC_ABS.Busy THEN 
		abs_do:=FALSE;
		MoveAbsExe:=FALSE;
	END_IF
MC_Jog(
	Axis:=ref , 
	JogForward:=jogF_do , 
	JogBackwards:=jogB_do , 
	Mode:=MC_JOGMODE_CONTINOUS , 
	Position:= , 
	Velocity:=Velo , 
	Acceleration:=Acceleration , 
	Deceleration:=Deceleration , 
	Jerk:=Jerk , 
	Done=> , 
	Busy=> , 
	Active=> , 
	CommandAborted=> , 
	Error=> , 
	ErrorID=> );
MC_VELO(
	Axis:=ref , 
	Execute:=velo_do , 
	Velocity:=Velo , 
	Acceleration:=Acceleration , 
	Deceleration:=Deceleration , 
	Jerk:=Jerk , 
	Direction:= , 
	BufferMode:= MC_Aborting, 
	Options:= , 
	InVelocity=> , 
	Busy=> , 
	Active=> , 
	CommandAborted=> , 
	Error=> , 
	ErrorID=> );
	//IF MC_VELO.Busy THEN 
	//	velo_do:=FALSE;
	//END_IF
MC_stop(
	Axis:=ref , 
	Execute:=stop_do , 
	Deceleration:=Deceleration , 
	Jerk:=Jerk , 
	Options:= , 
	Done=> , 
	Busy=> , 
	Active=> , 
	CommandAborted=> , 
	Error=> , 
	ErrorID=> );
IF MC_stop.Done THEN 
	stop_do:=FALSE;
END_IF
END_ACTION

ACTION JOG:
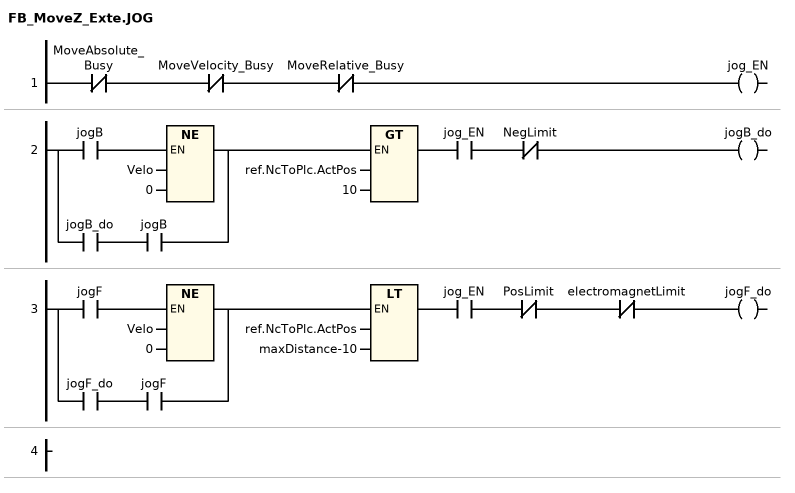
// NETWORK 1
jog_EN := NOT MoveAbsolute_Busy AND NOT MoveVelocity_Busy AND NOT MoveRelative_Busy;

// NETWORK 2
jogB_do := ((jogB AND Velo <> 0 OR jogB_do AND jogB) AND ref.NcToPlc.ActPos > 10) AND jog_EN AND NOT NegLimit;

// NETWORK 3
jogF_do := ((jogF AND Velo <> 0 OR jogF_do AND jogF) AND ref.NcToPlc.ActPos < (maxDistance-10)) AND jog_EN AND NOT PosLimit AND NOT electromagnetLimit;

// NETWORK 4
END_ACTION

ACTION MoveAbsolute:
(****************ABS********************)
R_TRIG2(CLK:=MoveAbsExe AND Ref.Status.NotMoving    , Q=> );

CASE step2 OF 
	0:				
		IF R_TRIG2.Q THEN 
			R_TRIG2(CLK:=FALSE);			
			MoveAbsExe:=FALSE;
			electromagnet_power:=FALSE;
			step2:=1;
		END_IF
	1:	
		IF   Velo<>0 THEN 		
			abs_do:=TRUE;
			step2:=2;
		END_IF
	2:
		IF MC_ABS.Busy THEN 
			abs_do:=FALSE;								
			step2 :=0;
		END_IF	
END_CASE


IF  MoveAbsolute_Busy THEN 
	MoveRelExe:=FALSE;
	MoveVelocityExe:=FALSE;
	electromagnet_power:=FALSE;
END_IF
END_ACTION

ACTION MoveRelative:
(****************Rel********************)
R_TRIG1(CLK:=MoveRelExe AND Ref.Status.NotMoving   , Q=> );
CASE step1 OF 
	0:				
		IF R_TRIG1.Q THEN 
			R_TRIG1(CLK:=FALSE);
			MoveRelExe:=FALSE;
			electromagnet_power:=FALSE;
			step1:=1;
		END_IF
	1:	
		IF TargetRel <>0 AND Velo<>0 THEN 		
			rel_do:=TRUE;
			step1:=2;
		END_IF
	2:
		IF MC_REL.Busy THEN 
			rel_do:=FALSE;								
			step1 :=0;
		END_IF	
END_CASE

IF MoveRelative_Busy THEN 
	MoveAbsExe:=FALSE;
	MoveVelocityExe:=FALSE;
	electromagnet_power:=FALSE;
END_IF
END_ACTION

ACTION MoveVelocity:
(****************当做自动测高********************)
IF electromagnetLimit THEN 
	MoveVelocityExe:=FALSE;
END_IF
R_TRIG3(CLK:=MoveVelocityExe AND Ref.Status.NotMoving AND NOT electromagnetLimit  , Q=> );
CASE step3 OF 
	0:				
		IF R_TRIG3.Q THEN 
			R_TRIG3(CLK:=FALSE);
			MoveVelocityExe:=FALSE;
			velo_do:=FALSE;		
			step3:=1;
		END_IF
	1:	//电磁铁得电
		electromagnet_power:=TRUE;
		IF   Velo<>0 THEN 		
			velo_do:=TRUE;
			step3:=2;
		END_IF
		
	2:	//碰到电磁铁，停止
		IF electromagnetlimit THEN 
			electromagnet_power:=FALSE;
			velo_do:=FALSE;
			stop_do:=TRUE;
			step3 :=0;
		END_IF
END_CASE
MoveVelocity_Busy:=MC_VELO.Busy ;

IF MoveVelocity_Busy THEN 
	MoveRelExe:=FALSE;
	MoveAbsExe:=FALSE;
END_IF
END_ACTION

END_FUNCTION_BLOCK

// ---- POUs/030_MediaTransport/UpDownSlot/FB/FB_UpDownSlotS1.TcPOU
FUNCTION_BLOCK FB_UpDownSlotS1
VAR_INPUT	
	timeout_up			:LREAL;//MS
	timeout_down		:LREAL;//MS
	extra_down_time		:LREAL;//Ms
	sensor_up			:BOOL;
	sensor_down			:ARRAY[1..16] OF BOOL;

END_VAR
VAR_OUTPUT
	MoveDown_do			:BOOL;
	MoveUp_do			:BOOL;
	Break					:BOOL;//启动提前，停止延后
	anysensor_down		:BOOL;
	state				:INT;
	error_code				:INT;
	error				:BOOL;
END_VAR
VAR
	step				:INT;
	Ton_MoveUp_do		:Tc2_Standard.TON;
	Ton_MoveDown_do		:Tc2_Standard.TON;
	Ton_MoveDown_delay_do :TON;
	ET_Ton_MoveUp_do	:LREAL;
	ET_Ton_MoveDown_do	:LREAL;
	
	i: INT;
	dely_ton_on:Tc2_Standard.TON;//启动时
	dely_ton_off:Tc2_Standard.TON;//关断时
	dely_time:TIME:=T#10MS;
	F_trig_move:Tc2_Standard.F_TRIG;
	en_ton:BOOL;
END_VAR
VAR_IN_OUT
	Initialize			:BOOL;
	MoveDown			:BOOL;
	MoveUp				:BOOL;
	SetOff				:BOOL;
END_VAR

ET_Ton_MoveUp_do:=TIME_TO_LREAL(Ton_MoveUp_do.ET);
ET_Ton_MoveDown_do:=TIME_TO_LREAL(Ton_MoveDown_do.ET);

FOR i:=1 TO 16 DO 
	IF sensor_down[i] THEN 
		anysensor_down:=TRUE;
		EXIT;
	ELSE 
		anysensor_down:=FALSE;
	END_IF
END_FOR

CASE step OF
0://waiting
	IF Initialize THEN 
		step:=5;
	ELSIF MoveDown THEN 
		step:=41;
	ELSIF MoveUp THEN 
		step:=71;
	ELSIF SetOff OR GVL.Reset THEN 
		step:=99;
	END_IF
5://0ff
	MoveDown:=FALSE;
	MoveUp:=FALSE;
	SetOff:=FALSE;
	MoveDown_do:=FALSE;
	MoveUp_do:=FALSE;
	Ton_MoveDown_do(IN:=FALSE , PT:= , Q=> , ET=> );
	Ton_MoveUp_do(IN:=FALSE , PT:= , Q=> , ET=> );
	
	state:=UpDownSlotStateEnum.off;
	error_code:=UpDownSlotErrorEnum.no_error;

	IF Initialize THEN 
		Initialize:=FALSE;		
		step:=10;
	END_IF
10://打开抱闸
	Initialize:=FALSE;
	Break:=TRUE;
	dely_ton_on(IN:=TRUE , PT:=dely_time , Q=> , ET=> );
	IF dely_ton_on.Q THEN 
		dely_ton_on(IN:=FALSE);
		step:=20;
	END_IF

20://初始化，执行上升指令	
	MoveUp_do:=TRUE;	
	MoveUp:=FALSE;
	step:=30;
30://waiting up
	state:=UpDownSlotStateEnum.waiting_up;
	Ton_MoveUp_do(IN:=TRUE , PT:=LREAL_TO_TIME(timeout_up) , Q=> , ET=> );
	IF 	ET_Ton_MoveUp_do>0 AND ET_Ton_MoveUp_do<timeout_up THEN
		IF  sensor_up THEN 			
			MoveUp_do:=FALSE;
			state:=UpDownSlotStateEnum.up;
			Ton_MoveUp_do(IN:=FALSE);
			MoveUp:=FALSE;
			step:=40;				
		END_IF
	ELSIF ET_Ton_MoveUp_do>=timeout_up   THEN 
		IF NOT sensor_up  THEN 
			error_code:=UpDownSlotErrorEnum.timeout_up;
			step:=100;
		END_IF
	END_IF
40://up	
	IF MoveDown  THEN 		
		step:=41;
	END_IF
	(************抱闸***********************)
	dely_ton_off(IN:=TRUE , PT:=dely_time , Q=> , ET=> );
		IF dely_ton_off.Q THEN 
			dely_ton_off(IN:=FALSE);
			Break:=FALSE;
			step:=0;
		END_IF
41://释放抱闸状态		
		IF MoveDown THEN 
			dely_ton_on(IN:=TRUE  , PT:=dely_time , Q=> , ET=> );
			Break:=TRUE;
			IF dely_ton_on.Q THEN 
				dely_ton_on(IN:=FALSE);						
				step:=50;
			END_IF	
		END_IF
50://waiting down
	MoveDown_do:=TRUE;
	MoveDown:=FALSE;
	state:=UpDownSlotStateEnum.waiting_down;
	
	Ton_MoveDown_do(IN:=TRUE , PT:=LREAL_TO_TIME(timeout_down) , Q=> , ET=> );
	IF 	ET_Ton_MoveDown_do>0 AND ET_Ton_MoveDown_do<timeout_down THEN		
		IF  anysensor_down AND NOT sensor_up THEN 
			step:=51;				
		END_IF
	ELSIF ET_Ton_MoveDown_do>=timeout_down  THEN 
		IF NOT  anysensor_down  THEN 
			error_code:=UpDownSlotErrorEnum.timeout_down;
			step:=100;
		END_IF
	END_IF
51://DELAY_DOWN
	Ton_MoveDown_do(IN:=FALSE);
	Ton_MoveDown_delay_do(IN:=TRUE , PT:=LREAL_TO_TIME(extra_down_time) , Q=> , ET=> );
	IF Ton_MoveDown_delay_do.Q THEN 
		Ton_MoveDown_delay_do(IN:=FALSE);
		MoveDown_do:=FALSE;
		state:=UpDownSlotStateEnum.down;
		MoveDown:=FALSE;
		step:=60;	
	END_IF		
	
60://down
	IF MoveUp  THEN 
		step:=20;	
	END_IF
	
	(************抱闸***********************)
	dely_ton_off(IN:=TRUE , PT:=dely_time , Q=> , ET=> );
		IF dely_ton_off.Q THEN 
			dely_ton_off(IN:=FALSE);
			Break:=FALSE;
			step:=0;	
		END_IF	
71://释放 抱闸状态		
		IF MoveUp THEN 
			Break:=TRUE;
			dely_ton_on(IN:=TRUE  , PT:=dely_time , Q=> , ET=> );
			IF dely_ton_on.Q THEN 
				dely_ton_on(IN:=FALSE);							
				step:=20;
			END_IF	
		END_IF
99://setoff
	SetOff:=FALSE;
	error:=FALSE;
	Break:=FALSE;
	MoveDown:=FALSE;
	MoveUp:=FALSE;	
	Initialize:=FALSE;
	MoveDown_do:=FALSE;
	MoveUp_do:=FALSE;
	Ton_MoveDown_do(IN:=FALSE , PT:= , Q=> , ET=> );
	Ton_MoveUp_do(IN:=FALSE , PT:= , Q=> , ET=> );	
	state:=UpDownSlotStateEnum.off;
	error_code:=UpDownSlotErrorEnum.no_error;
	step:=0;
100://error
	error:=TRUE;
	state:=UpDownSlotStateEnum.error;
	MoveUp_do:=FALSE;
	MoveDown_do:=FALSE;
	Break:=FALSE;
	step:=0;	
END_CASE

(************setoff***********************)
IF SetOff OR GVL.Reset THEN 
	step:=99;
END_IF
IF state<>UpDownSlotStateEnum.off AND state<>UpDownSlotStateEnum.error AND  GVL.Emstop_Button THEN 
	error_code:=UpDownSlotErrorEnum.emergency_error;
	step:=100;
END_IF

END_FUNCTION_BLOCK

// ---- POUs/030_MediaTransport/UpDownSlot/FB/FB_UpDownSlotS2_S6.TcPOU
FUNCTION_BLOCK FB_UpDownSlotS2_S6
VAR_INPUT	
	timeout_up			:LREAL:=5000;//MS
	timeout_down		:LREAL:=5000;//MS
	sensor_up			:BOOL;

END_VAR
VAR_OUTPUT
	MoveDown_do			:BOOL;
	MoveUp_do			:BOOL;
	
	state				:INT;
	error_code				:INT;
	error				:BOOL;
END_VAR
VAR
	step				:INT;
	Ton_MoveUp_do		:Tc2_Standard.TON;
	Ton_MoveDown_do		:Tc2_Standard.TON;
	ET_Ton_MoveUp_do	:LREAL;
	ET_Ton_MoveDown_do	:LREAL;

END_VAR
VAR_IN_OUT
	Initialize			:BOOL;
	MoveDown			:BOOL;
	MoveUp				:BOOL;
	SetOff				:BOOL;
END_VAR

ET_Ton_MoveUp_do:=TIME_TO_LREAL(Ton_MoveUp_do.ET);
ET_Ton_MoveDown_do:=TIME_TO_LREAL(Ton_MoveDown_do.ET);


CASE step OF
0://waiting
	IF Initialize THEN 
		step:=5;
	ELSIF MoveDown THEN 
		step:=40;
	ELSIF MoveUp THEN 
		step:=60;
	ELSIF SetOff OR GVL.Reset THEN 
		step:=99;
	END_IF
5://0ff
	MoveDown:=FALSE;
	MoveUp:=FALSE;
	SetOff:=FALSE;
	MoveDown_do:=FALSE;
	MoveUp_do:=FALSE;
	Ton_MoveDown_do(IN:=FALSE , PT:= , Q=> , ET=> );
	Ton_MoveUp_do(IN:=FALSE , PT:= , Q=> , ET=> );
	
	state:=UpDownSlotStateEnum.off;
	error_code:=UpDownSlotErrorEnum.no_error;

	IF Initialize THEN 
		Initialize:=FALSE;
		IF timeout_up>0 AND timeout_down>0  THEN 
			step:=10;
		END_IF
	END_IF
10://
	timeout_up:=5000;(*Initialize时，未给timeout，先赋值一下*)
	Initialize:=FALSE;
	step:=20;
20://初始化，执行上升指令	
	MoveUp_do:=TRUE;	
	MoveUp:=FALSE;
	step:=30;
30://waiting up
	state:=UpDownSlotStateEnum.waiting_up;
	Ton_MoveUp_do(IN:=TRUE , PT:=LREAL_TO_TIME(timeout_up) , Q=> , ET=> );
	IF 	ET_Ton_MoveUp_do>0 AND ET_Ton_MoveUp_do<timeout_up THEN
		IF  sensor_up THEN 
			Ton_MoveUp_do(IN:=FALSE);
			MoveUp_do:=FALSE;
			state:=UpDownSlotStateEnum.up;			
			MoveUp:=FALSE;
			step:=0;		
		END_IF
	ELSIF ET_Ton_MoveUp_do>=timeout_up  THEN 
		IF NOT sensor_up  THEN 
			error_code:=UpDownSlotErrorEnum.timeout_up;
			step:=100;
		END_IF
	END_IF
40://up
	MoveUp:=FALSE;
	IF MoveDown THEN 
		MoveDown_do:=TRUE;
		step:=50;
	END_IF
50://waiting down
	MoveDown:=FALSE;
	state:=UpDownSlotStateEnum.waiting_down;
	
	Ton_MoveDown_do(IN:=TRUE , PT:=LREAL_TO_TIME(timeout_down) , Q=> , ET=> );
	IF ET_Ton_MoveDown_do>=timeout_down THEN
		Ton_MoveDown_do(IN:=FALSE);
		MoveDown_do:=FALSE;
		state:=UpDownSlotStateEnum.down;
		step:=0;	
	END_IF
60://down
	MoveDown:=FALSE;
	IF MoveUp THEN 
		step:=20;
	END_IF
99://setoff
	SetOff:=FALSE;
	error:=FALSE;
	MoveDown:=FALSE;
	MoveUp:=FALSE;
	Initialize:=FALSE;
	MoveDown_do:=FALSE;
	MoveUp_do:=FALSE;
	Ton_MoveDown_do(IN:=FALSE , PT:= , Q=> , ET=> );
	Ton_MoveUp_do(IN:=FALSE , PT:= , Q=> , ET=> );	
	state:=UpDownSlotStateEnum.off;
	error_code:=UpDownSlotErrorEnum.no_error;
	step:=0;
100://error
	error:=TRUE;
	state:=UpDownSlotStateEnum.error;
	MoveUp_do:=FALSE;
	MoveDown_do:=FALSE;
	step:=0;
		
END_CASE
(************setoff***********************)
IF SetOff OR GVL.Reset THEN 	
	step:=99;
END_IF
IF state<>UpDownSlotStateEnum.off  AND state<>UpDownSlotStateEnum.error AND GVL.Emstop_Button THEN 
	error_code:=UpDownSlotErrorEnum.emergency_error;
	step:=100;
END_IF

END_FUNCTION_BLOCK

// ---- POUs/040_System/FootPedal/FB/FB_FootPedal.TcPOU
FUNCTION_BLOCK FB_FootPedal
VAR_INPUT
	PedalPressed1			:BOOL;	
	PedalPressed2			:BOOL;
	PedalPressed3			:BOOL;
	debounce_time			:LREAL;//ms The amount of time that the foot pedal does not register another click.	
END_VAR
VAR_OUTPUT
	error_code					:INT;	//	
	state					:INT;	//	
	pressed					:INT;//‘none’, ‘pedal1’, ‘pedal2’, ‘pedal3’	
	Error					:BOOL;
END_VAR
VAR
	ton1:Tc2_Standard.TON;
	step:INT;
	TRIG1:Tc2_Standard.R_TRIG;
END_VAR
VAR_IN_OUT
	Reset					:BOOL;
END_VAR

CASE step OF
0:
	state:=FootPedalStateEnum.ready;
	error_code:=FootPedalErrorEnum.no_error;
	pressed:=0;
	ton1(IN:=FALSE);
	Reset:=FALSE;
	
	IF PedalPressed1 THEN 
		step:=10;
	ELSIF PedalPressed2 THEN 
		step:=20;
	ELSIF PedalPressed3 THEN 
		step:=30;
	END_IF
	
10:	
	IF PedalPressed1 THEN 
		pressed:=1;
	ELSE 
		pressed:=0;
		step:=50;
	END_IF
	
20:	
	IF PedalPressed2 THEN 
		pressed:=2;
	ELSE 
		pressed:=0;
		step:=50;
	END_IF

30:	
	IF PedalPressed3 THEN 
		pressed:=3;
	ELSE 
		pressed:=0;
		step:=50;
	END_IF

50://缓冲
	ton1(IN:=TRUE , PT:=LREAL_TO_TIME(debounce_time) , Q=> , ET=> );
	IF ton1.Q THEN 
		step:=0;
	END_IF
100://error
	state:=FootPedalStateEnum.error;
	pressed:=0;
	error:=TRUE;
	IF Reset OR GVL.Reset THEN 
		Reset:=FALSE;
		error:=FALSE;
		step:=0;
	END_IF
END_CASE

IF Reset OR GVL.Reset THEN 
	Reset:=FALSE;
	error:=FALSE;
	step:=0;
END_IF


TRIG1(CLK:=GVL.Emstop_Button , Q=> ); 
	IF TRIG1.Q THEN 
		error_code:=FootPedalErrorEnum.emergency_error;
		step:=100;
	END_IF

END_FUNCTION_BLOCK

// ---- POUs/040_System/SystemEnvironment/FB/FB_SystemEnvironment.TcPOU
FUNCTION_BLOCK FB_SystemEnvironment
VAR_INPUT
	IO_Error				:BOOL;

	duration:LREAL;//S
	period :LREAL;//S
END_VAR
VAR_OUTPUT
	temp_measured:LREAL;
	humidity_measured:LREAL;
	bqbuzzer:BOOL;
	Error:BOOL;
END_VAR
VAR
	step:INT;
	FB_Buzzer:FB_Buzzer;
	Start_Exe:BOOL;
END_VAR
VAR_IN_OUT
	error_code			:INT;
	state							:INT;
	Reset:BOOL;
	BuzzerOn				:BOOL;
	BuzzerOff				:BOOL;
END_VAR

CASE step OF
0://ready
	Reset:=FALSE;
	state:=EnvironmentStateEnum.ready;
	error_code:=EnvironmentErrorEnum.no_error;
	temp_measured:=GVL.temp_measured;
	humidity_measured:=GVL.humidity_measured;
	//IF IO_Error THEN
		//step:=100;
	//END_IF
	IF BuzzerOn AND NOT BuzzerOff THEN 
		BuzzerOn:=FALSE;
		Start_Exe:=TRUE;
	ELSIF BuzzerOff AND NOT BuzzerOn THEN 
		Start_Exe:=FALSE;
		BuzzerOff:=FALSE;
	END_IF
	
	FB_Buzzer(duration:=duration , period:=period , bqbuzzer=>bqbuzzer , Start_Exe:=Start_Exe );
99://setoff	
		Reset:=FALSE;
		error_code:=EnvironmentErrorEnum.no_error;
		state:=EnvironmentStateEnum.ready;
		error:=FALSE;
		step:=0;
100://error
	state:=EnvironmentStateEnum.error;	
	error:=TRUE;
	IF Reset OR GVL.Reset THEN 
		step:=99;
	END_IF
END_CASE

IF Reset OR GVL.Reset THEN 
		step:=99;
END_IF

IF state<>EnvironmentStateEnum.error THEN 
	IF GVL.Emstop_Button THEN 
		error_code:=EnvironmentErrorEnum.emergency_error;
		step:=100;
	ELSIF IO_Error THEN
		error_code:=EnvironmentErrorEnum.unknown_error;
		step:=100;
	END_IF
END_IF

END_FUNCTION_BLOCK

// ---- POUs/050_InkSystem/ISS/P_ISS.TcPOU
PROGRAM P_ISS
VAR

	i:INT;

	log_ErrorEnum:ISSErrorEnum;
	log_ID:INT;
	LC,LM,Y,M,C,K,W,F,P:INT;
	setoff_trig:ARRAY[1..9] OF Tc2_Standard.R_TRIG;
END_VAR

ACT_LED_Level();
ACT_LOG();
LC:=1; LM:=2;Y:=3;M:=4;C:=5;K:=6;W:=7;F:=8;P:=9;

FOR i:=1 TO 9 DO
	IF GVL_API.stISS[i].Initialize THEN 
		GVL_API.stISS[i].Initialize:=FALSE;
	END_IF
	IF GVL_API.stISS[i].Setoff OR GVL.Reset THEN 
		GVL_API.stISS[i].Setoff:=FALSE;
	END_IF
END_FOR

ACTION ACT_LED_Level:
(*******************led***************************)	
FOR i:=1 TO 9 DO 
	stOutput .bqsensor_blink[i]:=GVL_API.stISS[i].sensor_blink;			//LC,LM,Y,M,C,K,W,F,P
																		
END_FOR

FOR i:=1 TO 9 DO 
	setoff_trig[i](CLK:=GVL_API.stISS[i].Setoff , Q=> );
	IF setoff_trig[i].Q THEN 
		stOutput .bqsensor_blink[i]:=GVL_API.stISS[i].sensor_blink:=FALSE;	
	END_IF
END_FOR


(**********废液LED**************)
IF GVL.MainTankLevel[10]>=3 THEN 
	stOutput .bqsensor_blink[10]:=TRUE;
ELSE
	stOutput .bqsensor_blink[10]:=FALSE;
END_IF

(*******************mainlevel***************************)	
FOR i:=1 TO 9 DO 
	GVL_API.stISS[i].mainTankLevel:=GVL.MainTankLevel[i];
END_FOR
END_ACTION

ACTION ACT_LOG:
(*************************LOG*******************************************)
log_ID:=500;
//ISS1  501-505
//ISS2  506-510
//ISS3  511-515
//ISS4  516-520
//ISS5  521-525
//ISS6  526-530
//ISS7  531-535
//ISS8  536-540
//ISS9  540-545
FOR i:=1 TO 9 DO 
//Initialize 
AlarmActionArray[log_ID+5*(i-1)+1].AlarmMsg.EN	:=	CONCAT('ISS',INT_TO_STRING(i));
AlarmActionArray[log_ID+5*(i-1)+1].AlarmMsg.EN	:=CONCAT(AlarmActionArray[log_ID+5*(i-1)+1].AlarmMsg.EN,
																				' Initialize');																			
fbSetAlarm[log_ID+5*(i-1)+1](
	InUse:=TRUE , 
	EventId:=log_ID+5*(i-1)+1 , 
	EventActive:=GVL_API.stISS[i].Initialize , 
	EventClass:=Alm_EventClass.Event , 
	ToTheLogFile:=TRUE, 
	ToTheHistory:=TRUE , 
 );
 
 //ERROR,log_ErrorEnum只能等于一个常数,   
CASE GVL_API.stISS[i].error_code  OF
0	:	log_ErrorEnum	:=	0	;
1	:	log_ErrorEnum	:=	1	;
2	:	log_ErrorEnum	:=	2	;
4	:	log_ErrorEnum	:=	4	;
6	:	log_ErrorEnum	:=	6	;
//7	:	log_ErrorEnum	:=	7	;
8	:	log_ErrorEnum	:=	8	;
9	:	log_ErrorEnum	:=	9	;
10	:	log_ErrorEnum	:=	10	;
666	:	log_ErrorEnum	:=	666	;

END_CASE
AlarmActionArray[log_ID+5*(i-1)+2].AlarmMsg.EN	:=	CONCAT('ISS',INT_TO_STRING(i));
AlarmActionArray[log_ID+5*(i-1)+2].AlarmMsg.EN	:=CONCAT(AlarmActionArray[log_ID+5*(i-1)+2].AlarmMsg.EN,' Error: ');	
AlarmActionArray[log_ID+5*(i-1)+2].AlarmMsg.EN	:=CONCAT(AlarmActionArray[log_ID+5*(i-1)+2].AlarmMsg.EN,
																				TO_STRING(log_ErrorEnum));	

fbSetAlarm[log_ID+5*(i-1)+2](
	InUse:=TRUE , 
	EventId:=log_ID+5*(i-1)+2 , 
	EventActive:=GVL_API.stISS[i].error_code<>0 AND GVL_API.stISS[i].error_code<>666 , 
	EventClass:=Alm_EventClass.Alarm , 
	ToTheLogFile:=TRUE, 
	ToTheHistory:=TRUE , 
 );
 

//Setoff
AlarmActionArray[log_ID+5*(i-1)+3].AlarmMsg.EN	:=	CONCAT('ISS',INT_TO_STRING(i));
AlarmActionArray[log_ID+5*(i-1)+3].AlarmMsg.EN	:=CONCAT(AlarmActionArray[log_ID+5*(i-1)+3].AlarmMsg.EN,
																				' Setoff');		
fbSetAlarm[log_ID+5*(i-1)+3](
	InUse:=TRUE , 
	EventId:=log_ID+5*(i-1)+3 , 
	EventActive:=GVL_API.stISS[i].Setoff   , 
	EventClass:=Alm_EventClass.Event , 
	ToTheLogFile:=TRUE, 
	ToTheHistory:=TRUE , 
 );
END_FOR

 (*************em-stop*     549**************
AlarmActionArray[549].AlarmMsg.EN	:='ISS Error:emergency_error';	
fbSetAlarm[549](
	InUse:=TRUE , 
	EventId:=549 , 
	EventActive:=GVL_API.stISS[1].error_code=666 , 
	EventClass:=Alm_EventClass.Alarm , 
	ToTheLogFile:=TRUE, 
	ToTheHistory:=TRUE , 
 );
*)
END_ACTION

END_PROGRAM

// ---- POUs/030_MediaTransport/P_MediaTransport.TcPOU
PROGRAM P_MediaTransport
VAR
END_VAR

P_TableVacuum();
P_UpDownSlot();

END_PROGRAM

// ---- POUs/010_Motion/MotionBase/PTP/Axis_IO.TcPOU
FUNCTION_BLOCK Axis_IO
VAR_INPUT
	snHome:			BOOL;(*原点*)
	snLimitP:		BOOL;(*正限*)
	snLimitN:		BOOL;(*负限*)
	snSpindle		:BOOL;	//z轴测高
	btManualJogF:	BOOL;(*点动按钮正*)
	btManualJogB:	BOOL;(*点动按钮负*)
	btManualABS:    BOOL;(*点动绝对*)
END_VAR

;

END_FUNCTION_BLOCK

// ---- POUs/070_RollToRoll/FB/FB_RollToRoll_Torque.TcPOU
(********************************)
FUNCTION_BLOCK FB_RollToRoll_Torque
VAR_INPUT
	biClamp_hold				:BOOL;
	Un_Rewinder					:BOOL;//false:unwinder;true:rewinder
	Max_velo					:LREAL;//r/min
	REF							:AXIS_REF;
	usable				        :BOOL;//
	acceleration				:LREAL;//
	deceleration				:LREAL;//
	rate						:DINT;// % 0-100 Motor speed or torque.
	untension_rate				:DINT:=10;//% Duty cycle for the motor speed during untensioning
	tension_mode				:BOOL;// Indicates the printside: ‘inside’ or ‘outside’ false:outside
	tension_timeout				:LREAL:=10;//ms
	untension_timeout			:LREAL:=5;//ms
	brake_timeout				:LREAL:=120;//MS
	
END_VAR
VAR_OUTPUT
	error_code					:UDINT;	//	
	state					:INT;	//
	Axis_ErrorId			:UDINT;
	Break_Power				:BOOL:=FALSE;
	Clutch_Out				:BOOL;
	out_rTorqueVelocityLimit        :LREAL;
	Initialized					:BOOL;
	error							:BOOL;
	tensioned					:BOOL;
	untensioned				:BOOL;
END_VAR
VAR
	step:INT;
	MC_POWER:MC_Power;
	MC_Read:MC_ReadStatus;
	MC_ABS:MC_MoveAbsolute;
	MC_REL:MC_MoveRelative;
	MC_Jog:MC_Jog;
	MC_Stop:MC_Stop;
	MC_Reset:Tc2_MC2.MC_Reset;
	MC_SetPos:Tc2_MC2.MC_SetPosition;
	mc_Torque:Tc2_MC2.MC_TorqueControl;
	
	power_do: BOOL;
	stop_do:BOOL;
	reset_do:BOOL;
	set_torque:LREAL;
	direction:MC_Direction;
	set_acceleration				:LREAL;//
	set_deceleration				:LREAL;//
	tension_ton:Tc2_Standard.TON;
	untension_ton:Tc2_Standard.TON;
	enbreak_ton:Tc2_Standard.TON;
	
	
	var_rTorque: LREAL;
	var_bTorqueCtrlExecute: BOOL;
	var_rTorqueRamp: LREAL := 100;
	
	ton1:Tc2_Standard.TON;
	F_trig_biClamp_hold:Tc2_Standard.F_TRIG;
END_VAR
VAR_IN_OUT
	Initialize					:BOOL;//
	SetActivate					:BOOL;//
	SetReady					:BOOL;//
	EnableBrake					:BOOL;//
	DisableBrake				:BOOL;
	StartTension				:BOOL;
	StopTension					:BOOL;
	Unlock						:BOOL;
	Lock						:BOOL;
	SetOff						:BOOL;
END_VAR

ACT_AXIS();
CASE step OF 
0://waiting	
	reset_do:=FALSE;
	
		IF Initialize THEN
			stop_do:=TRUE;
			step :=10;
		ELSIF SetActivate AND usable THEN 
			step :=20;
		ELSIF SetReady AND usable THEN 
			step :=30;
		ELSIF EnableBrake THEN 
			step :=30;
		ELSIF DisableBrake THEN 
			step :=40;
		ELSIF StartTension THEN 
			step :=30;
		ELSIF state=RTRStateEnum.tensioning AND  StopTension THEN 
			step :=50;
		ELSIF state=RTRStateEnum.tensioned AND  StopTension THEN 
			step :=60;
		END_IF
	
	IF  SetOff OR GVL.Reset THEN 
		step :=90;
	END_IF
	
	(***************状态自复位**************************)
	ton1(IN:=Initialized OR  tensioned OR untensioned , PT:=State_reset_time , Q=> , ET=> );
	IF ton1.Q THEN 
		Initialized:=FALSE;
		tensioned:=FALSE;
		untensioned:=FALSE;
	END_IF
10://Initializing
	Initialize:=FALSE;
	state:=RTRStateEnum.initializing;
	power_do :=TRUE;
	Break_Power:=FALSE;
	stop_do:=FALSE;
	IF rate>=0 AND  rate<=100  
	AND acceleration>0 AND deceleration>0 AND REF.Status.ControlLoopClosed THEN 
		 Initialized:=TRUE;
		 state:=RTRStateEnum.ready;
		step:=0;	
	END_IF
20://ready
	state:=RTRStateEnum.ready;
	SetReady:=FALSE;
	
	IF SetActivate THEN 
		SetActivate:=FALSE;
		Break_Power:=FALSE;
		state:=RTRStateEnum.active;
		step:=0;
	END_IF
30://active
	Break_Power:=FALSE;	
	untension_ton(IN:= FALSE);
	
	enbreak_ton(IN:=FALSE);
	IF SetReady THEN 
		SetReady:=FALSE;
		stop_do:=TRUE;
		state:=RTRStateEnum.ready;
		step:=0;
	END_IF
	
	IF NOT Un_Rewinder AND EnableBrake THEN //只有放卷有刹车				
		step:=40;
	END_IF
	
	IF StartTension AND tension_timeout>0 THEN 
		StartTension:=FALSE;
		state:=RTRStateEnum.tensioning;
		
		IF NOT  Un_Rewinder THEN 						//放卷
			IF tension_mode THEN 						//inside
				direction:=MC_Positive_Direction;
				var_rTorque:=rate;
			ELSE 										//outside
				direction:=MC_Negative_Direction;
				var_rTorque:=0-rate;
			END_IF
		ELSE											//收卷
			IF tension_mode THEN 						//inside
				direction:=MC_Negative_Direction;
				var_rTorque:=0-rate;
			ELSE 										//outside
				direction:=MC_Positive_Direction;
				var_rTorque:=rate;
			END_IF
		END_IF
		step:=50;
	END_IF
40://break_enable	
	IF EnableBrake THEN 
		EnableBrake:=FALSE;
		state:=RTRStateEnum.brake_enabled;
		Break_Power:=TRUE;	
		step:=0;			
	ELSIF DisableBrake THEN 
		DisableBrake:=FALSE;
		state:=RTRStateEnum.active;
		Break_Power:=FALSE;	
		enbreak_ton(IN:=FALSE);
		step:=0;
	END_IF	
50://tensioning
	var_bTorqueCtrlExecute:=TRUE;
	Clutch_Out:=TRUE;
	tension_ton(IN:=TRUE , PT:=LREAL_TO_TIME(tension_timeout) , Q=> , ET=> );
	IF tension_ton.Q   THEN 
		tensioned:=TRUE;
		state:=RTRStateEnum.tensioned;
		step:=0;
	END_IF
	IF StopTension THEN 
		StopTension:=FALSE;
		Clutch_Out:=FALSE;
		stop_do:=TRUE;
		state:=RTRStateEnum.untensioning;
		step:=70;
	END_IF
	
60://tensionde	
	tension_ton(IN:=FALSE);
	IF StopTension THEN 
		state:=RTRStateEnum.untensioning;
		StopTension:=FALSE;
		Clutch_Out:=FALSE;
		stop_do:=TRUE;
		step:=70;
	END_IF
70://untensionde
	untension_ton(IN:=TRUE , PT:= LREAL_TO_TIME(untension_timeout), Q=> , ET=> );
	IF untension_ton.Q THEN 
		untension_ton(IN:=FALSE);
		state:=RTRStateEnum.active;
		untensioned:=TRUE;
		step:=0;
	END_IF
90://setoff
	state:=RTRStateEnum.setting_off;
	
		SetOff:=FALSE;
		stop_do:=TRUE;
		reset_do:=TRUE;
		power_do:=FALSE;
		var_bTorqueCtrlExecute:=FALSE;
		Initialize:=FALSE;
		SetActivate:=FALSE;
		SetReady:=FALSE;
		EnableBrake:=FALSE;
		DisableBrake:=FALSE;
		StartTension:=FALSE;
		StopTension:=FALSE;
		error:=FALSE;
		
		Clutch_Out:=FALSE;
		enbreak_ton(IN:=FALSE);
		state:=RTRStateEnum.off;
		error_code:=RTRErrorEnum.no_error;
		step:=0;	
	
100://error
	state:=RTRStateEnum.error;
	error:=TRUE;
	stop_do:=FALSE;
	enbreak_ton(IN:=FALSE);
	step:=0;
	IF SetOff OR GVL.Reset THEN 
		step:=90;
	END_IF
END_CASE
IF SetOff OR GVL.Reset THEN 
		step:=90;
END_IF

(**************************ERROR**************************************************)
F_trig_biClamp_hold(CLK:=biClamp_hold , Q=> );
IF state<>RTRStateEnum.off  AND state<>RTRStateEnum.setting_off AND state<>RTRStateEnum.error THEN 
	IF GVL.Emstop_Button  THEN 	
		error_code:=RTRErrorEnum.emergency_error;
		stop_do:=TRUE;
		step:=100;
	ELSIF   REF.Status.Moving  AND  F_trig_biClamp_hold.Q THEN 	(*双卷动时，未检测到加紧,停止*)
		error_code:=RTRErrorEnum.roll_unclamped;			
		stop_do:=TRUE;
		step:=100;
	ELSIF Break_Power THEN 
		enbreak_ton(IN:=TRUE , PT:=LREAL_TO_TIME(brake_timeout) , Q=> , ET=> );
		IF enbreak_ton.Q THEN 
			error_code:=RTRErrorEnum.break_exceeded_timeout;
			step:=100;
		END_IF
	ELSIF MC_Read.ErrorID =18000 THEN 
		error_code:=RTRErrorEnum.Drive_not_ready_for_operation;
		stop_do:=TRUE;
		step:=100;
	ELSIF  MC_Read.ErrorID=17510 THEN 
		error_code:=RTRErrorEnum.Invalid_IO_data_for_more_than_n_subsequent_NC_cycles_encoder;
		stop_do:=TRUE;
		step:=100;	
	ELSIF  MC_Read.ErrorID <>0 THEN 
		error_code:=MC_Read.ErrorID;	
		stop_do:=TRUE;
		step:=100;
	END_IF
END_IF

